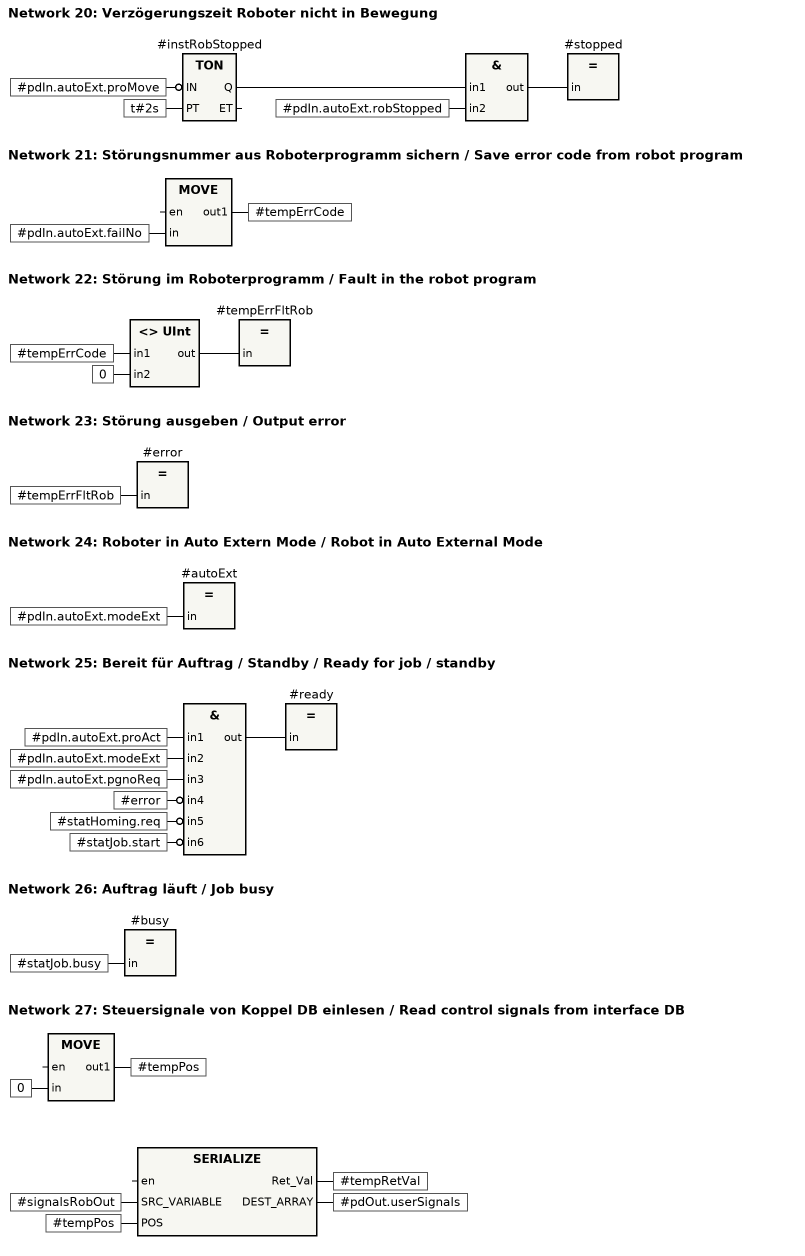
   #instRobStopped(IN := NOT #pdIn.autoExt.proMove, PT := t#2s);   // TON
   #stopped := #instRobStopped.Q AND #pdIn.autoExt.robStopped;
END_REGION

REGION Network 21: Störungsnummer aus Roboterprogramm sichern / Save error code from robot program
   #tempErrCode := #pdIn.autoExt.failNo;
END_REGION

REGION Network 22: Störung im Roboterprogramm / Fault in the robot program
   #tempErrFltRob := #tempErrCode <> 0;
END_REGION

REGION Network 23: Störung ausgeben / Output error
   #error := #tempErrFltRob;
END_REGION

REGION Network 24: Roboter in Auto Extern Mode / Robot in Auto External Mode
   #autoExt := #pdIn.autoExt.modeExt;
END_REGION

REGION Network 25: Bereit für Auftrag / Standby / Ready for job / standby
   #ready := #pdIn.autoExt.proAct AND #pdIn.autoExt.modeExt AND #pdIn.autoExt.pgnoReq AND NOT #error AND NOT #statHoming.req AND NOT #statJob.start;
END_REGION

REGION Network 26: Auftrag läuft / Job busy
   #busy := #statJob.busy;
END_REGION

REGION Network 27: Steuersignale von Koppel DB einlesen / Read control signals from interface DB
   // no SCL statement known for Serialize: written as a call
   #tempPos := 0;
   #tempRetVal := Serialize(SRC_VARIABLE := #signalsRobOut, POS := #tempPos, DEST_ARRAY => #pdOut.userSignals);
END_REGION

REGION Network 28: Peripherie schreiben / Write periphery
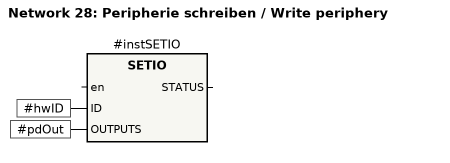
   #instSETIO(ID := #hwID, OUTPUTS := #pdOut);   // SETIO
END_REGION
END_FUNCTION_BLOCK

// folder: 9. Library/9.2 Actors/9.9.9 Simulation

FUNCTION_BLOCK "Actor2Ins2OutsSim"   // FB9991, FBD
TITLE = Aktoransteuerung 2 Ins / 2 Outs
{ S7_Optimized_Access := 'TRUE' }
VERSION : 0.1
// Ersteller: Andreas Fast Automation
// E-Mail: automation@fast-andreas.de
// 
// Projekt dient zu Demonstrationszwecken und frei genutzt werden.
// 
// Bausteinbeschreibung:
   VAR_INPUT
      iudtSimInterface : "typeSimInterface";
      ixHomePos : Bool;
      ixWorkPos : Bool;
   END_VAR
   VAR_IN_OUT
      qxHomePos : Bool;
      qxWorkPos : Bool;
      iqudtCtrl : Struct
         setHomePos : Bool;
         setWorkPos : Bool;
         isInHomePos : Bool;
         isInWorkPos : Bool;
      END_STRUCT;
      iqbSimIntAktor : Byte;   // Bit 0 = i_HomePos; Bit 1 = i_WorkPos; Bit 2 = q_SetHome; Bit 3 = q_SetWork
   END_VAR
   VAR
      sudtSimIntAktor : "typeSimAktor2Ins2Outs";
      sxSimDeactivatedFlag : Bool;
      sxSimDeactivated : Bool;
   END_VAR
   VAR_TEMP
      retVal : Int;
      tmpGrundstellungPhysikalisch : Bool;
      "tmpGrundstellungPhysikalisch+Virtuell" : Bool;
      tmpGrundstellungNurVirtuell : Bool;
   END_VAR
   VAR_TEMP   // added for the SCL form of the ladder/FBD networks
      _w1 : Bool;
      _w2 : Bool;
   END_VAR
BEGIN

REGION Network 1: Erkennung Simulation wird abgeschaltet
   // Wenn die Simulation abgeschaltet wird, sollen die physikalischen Ausgänge ihre aktuellen Zustände behalten um mögliche ungewollte Maschinenzustände zu vermeiden.
   // Das bedeutet, bei Abschaltung der Simulation werden die Ansteuerbefehle im "iqudtCtrl" and die physikalischen Ansteuerungen angepasst.
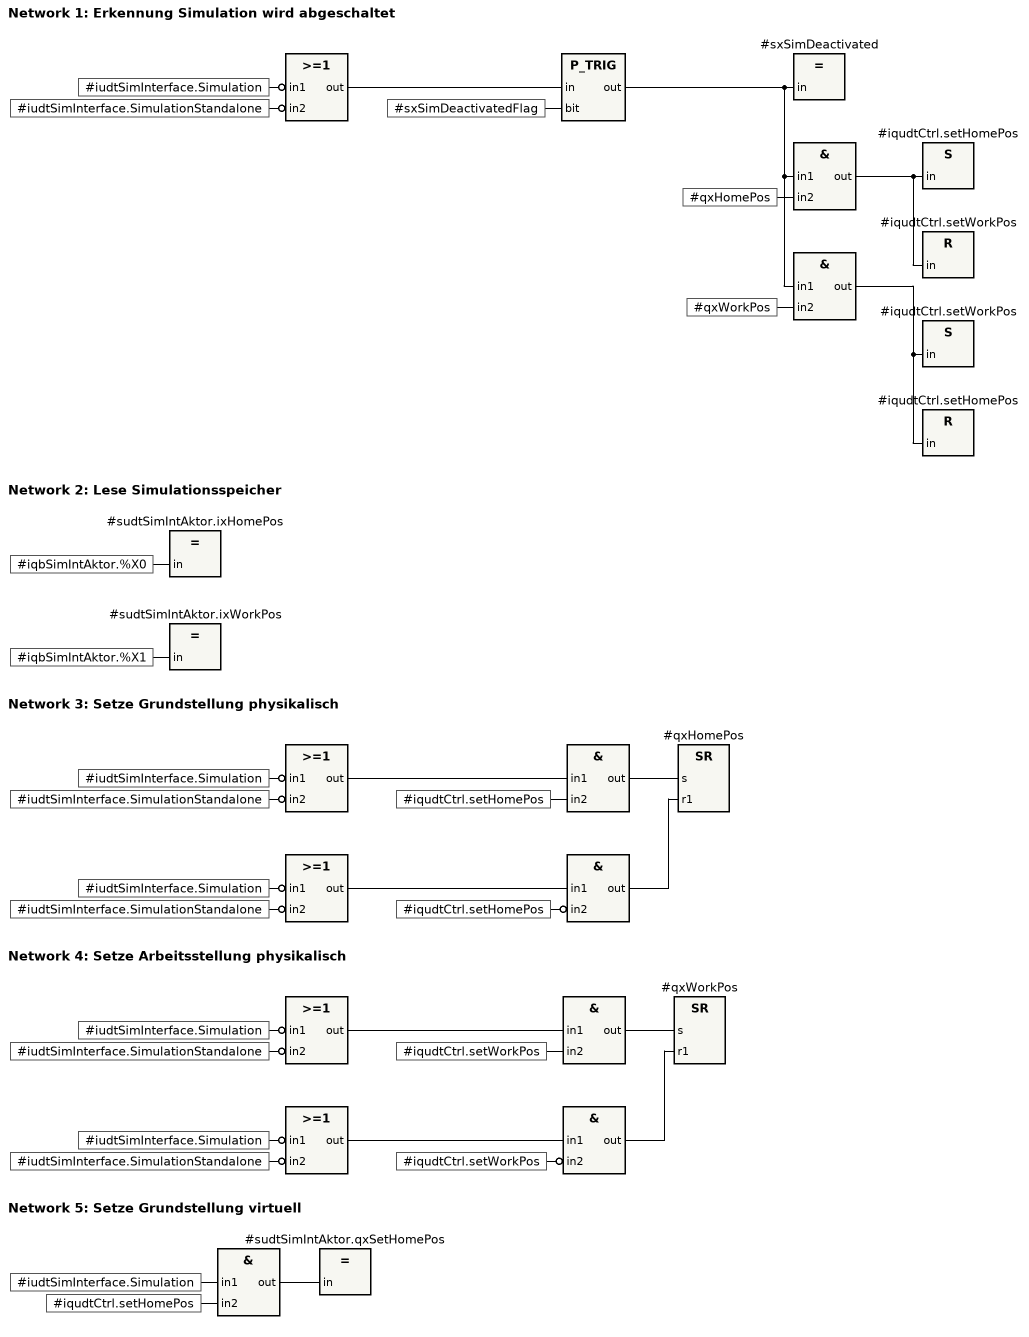
   #_w1 := NOT #iudtSimInterface.Simulation OR NOT #iudtSimInterface.SimulationStandalone;
   #_w2 := #_w1 AND NOT #sxSimDeactivatedFlag;   // rising edge
   #sxSimDeactivatedFlag := #_w1;
   #sxSimDeactivated := #_w2;
   IF #_w2 AND #qxHomePos THEN
       #iqudtCtrl.setHomePos := TRUE;
       #iqudtCtrl.setWorkPos := FALSE;
   END_IF;
   IF #_w2 AND #qxWorkPos THEN
       #iqudtCtrl.setWorkPos := TRUE;
       #iqudtCtrl.setHomePos := FALSE;
   END_IF;
END_REGION

REGION Network 2: Lese Simulationsspeicher
   #sudtSimIntAktor.ixHomePos := #iqbSimIntAktor.%X0;
   #sudtSimIntAktor.ixWorkPos := #iqbSimIntAktor.%X1;
END_REGION

REGION Network 3: Setze Grundstellung physikalisch
   IF (NOT #iudtSimInterface.Simulation OR NOT #iudtSimInterface.SimulationStandalone) AND #iqudtCtrl.setHomePos THEN
       #qxHomePos := TRUE;   // SR flip-flop
   END_IF;
   IF (NOT #iudtSimInterface.Simulation OR NOT #iudtSimInterface.SimulationStandalone) AND NOT #iqudtCtrl.setHomePos THEN
       #qxHomePos := FALSE;
   END_IF;
END_REGION

REGION Network 4: Setze Arbeitsstellung physikalisch
   IF (NOT #iudtSimInterface.Simulation OR NOT #iudtSimInterface.SimulationStandalone) AND #iqudtCtrl.setWorkPos THEN
       #qxWorkPos := TRUE;   // SR flip-flop
   END_IF;
   IF (NOT #iudtSimInterface.Simulation OR NOT #iudtSimInterface.SimulationStandalone) AND NOT #iqudtCtrl.setWorkPos THEN
       #qxWorkPos := FALSE;
   END_IF;
END_REGION

REGION Network 5: Setze Grundstellung virtuell
   #sudtSimIntAktor.qxSetHomePos := #iudtSimInterface.Simulation AND #iqudtCtrl.setHomePos;
END_REGION

REGION Network 6: Setze Arbeitsstellung virtuell
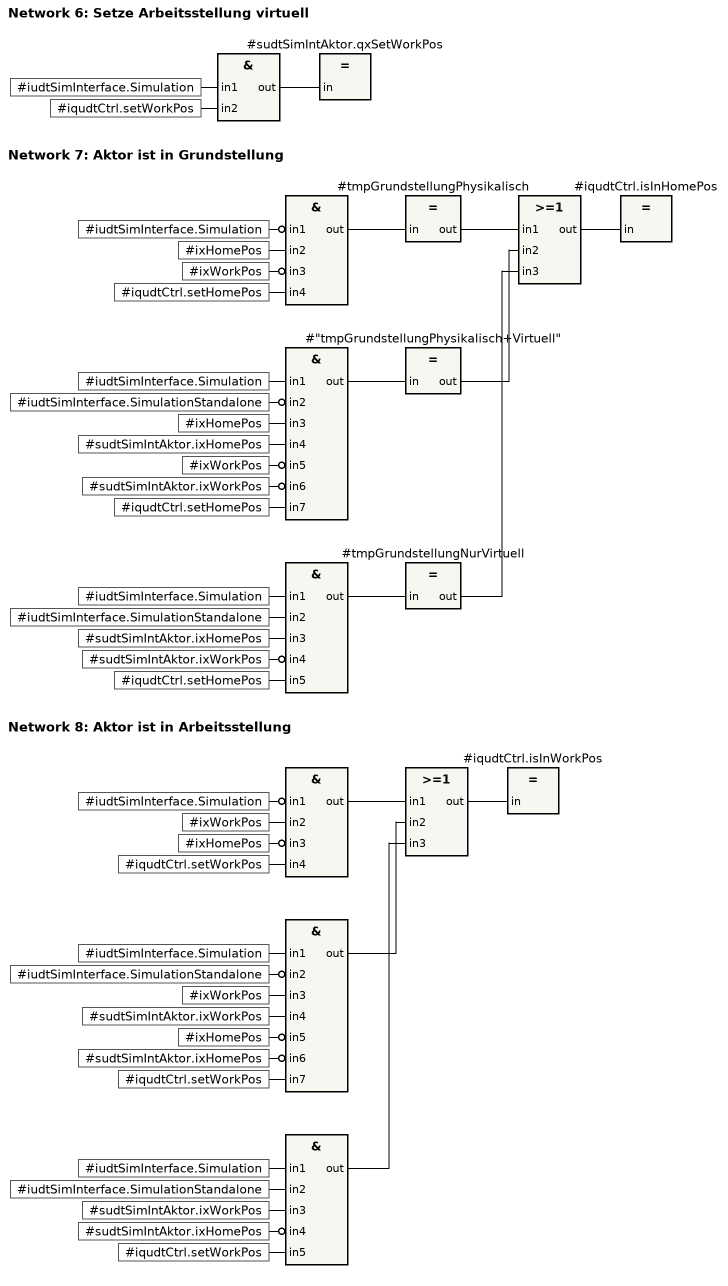
   #sudtSimIntAktor.qxSetWorkPos := #iudtSimInterface.Simulation AND #iqudtCtrl.setWorkPos;
END_REGION

REGION Network 7: Aktor ist in Grundstellung
   #tmpGrundstellungPhysikalisch := NOT #iudtSimInterface.Simulation AND #ixHomePos AND NOT #ixWorkPos AND #iqudtCtrl.setHomePos;
   #"tmpGrundstellungPhysikalisch+Virtuell" := #iudtSimInterface.Simulation AND NOT #iudtSimInterface.SimulationStandalone AND #ixHomePos AND #sudtSimIntAktor.ixHomePos AND NOT #ixWorkPos AND NOT #sudtSimIntAktor.ixWorkPos AND #iqudtCtrl.setHomePos;
   #tmpGrundstellungNurVirtuell := #iudtSimInterface.Simulation AND #iudtSimInterface.SimulationStandalone AND #sudtSimIntAktor.ixHomePos AND NOT #sudtSimIntAktor.ixWorkPos AND #iqudtCtrl.setHomePos;
   #iqudtCtrl.isInHomePos := #tmpGrundstellungPhysikalisch OR #"tmpGrundstellungPhysikalisch+Virtuell" OR #tmpGrundstellungNurVirtuell;
END_REGION

REGION Network 8: Aktor ist in Arbeitsstellung
   #iqudtCtrl.isInWorkPos := (NOT #iudtSimInterface.Simulation AND #ixWorkPos AND NOT #ixHomePos AND #iqudtCtrl.setWorkPos) OR (#iudtSimInterface.Simulation AND NOT #iudtSimInterface.SimulationStandalone AND #ixWorkPos AND #sudtSimIntAktor.ixWorkPos AND NOT #ixHomePos AND NOT #sudtSimIntAktor.ixHomePos AND #iqudtCtrl.setWorkPos) OR (#iudtSimInterface.Simulation AND #iudtSimInterface.SimulationStandalone AND #sudtSimIntAktor.ixWorkPos AND NOT #sudtSimIntAktor.ixHomePos AND #iqudtCtrl.setWorkPos);
END_REGION

REGION Network 9: Schreibe Aktorbefehle zur Simulation
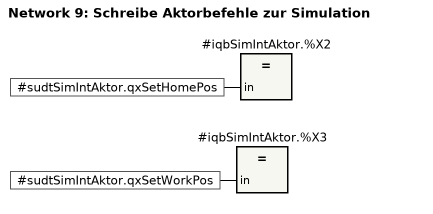
   #iqbSimIntAktor.%X2 := #sudtSimIntAktor.qxSetHomePos;
   #iqbSimIntAktor.%X3 := #sudtSimIntAktor.qxSetWorkPos;
END_REGION
END_FUNCTION_BLOCK

// folder: 9. Library/9.3 Processes

FUNCTION_BLOCK "Process_Stopper"   // FB9301, FBD
TITLE = Steuerung eines Stoppers
{ S7_Optimized_Access := 'TRUE' }
VERSION : 0.1
   VAR_INPUT
      ixBypass : Bool;   // UP umgehen / beenden
      ixStopperClosed : Bool;   // Stopper ist geschlossen/oben
      ixCarrierPresent : Bool;   // WT am Stopper vorhanden
      ixTargetReached : Bool := true;   // WT-Sensor des nächsten Ziels (falls nicht vorhanden muss dieser Eingang "true" sein)
      ixStop : Bool;   // Stoppt Ablauf / Schließt wieder den Stopper (z.B. bei einer Störung ausserhalb)
      itStopperRelease : Time := T#50ms;   // Zusätzliche Verzögerungszeit für Stopper öffnen, nachdem WT den Stopper verlassen hat
      itMaxRuntime : Time := t#5s;   // Maximale Laufzeit für diesen Prozess
   END_VAR
   VAR_OUTPUT
      qxSeqActive : Bool;   // Stopperablauf ist aktiv
      qxIsInHome : Bool;   // Ist in Grundstellung
      qxStopperOpen : Bool;   // Stopper öffnen
      qxError : Bool;   // Sammelstörung
      qbErrorCode : Byte;   // Ausgabe Fehlercode (siehe Sammelstörung Netzwerkkommentar)
   END_VAR
   VAR_IN_OUT
      signals : "typeStationSignals";   // Stationssignale
      iqxRequest : Bool;   // 1 = Starte Ablauf (wird nach Ausführung intern zurückgesetzt)
   END_VAR
   VAR
      sinstTonStopperOpened : TON_TIME;
      sinstTonStopperBusyError : TON_TIME;
      sinstTonMaxRuntime : TON_TIME;
      sxStep1 : Bool;
      sxStep2 : Bool;
      sxStep3 : Bool;
      sxCheckWtIsGone : Bool;   // Prüfe, ob WT den Stopper verlassen hat
   END_VAR
   VAR_TEMP
      txWT_Error_1 : Bool;
      txWT_Error_2 : Bool;
      txWT_Error_3 : Bool;
      txWT_Error_4 : Bool;
      txWT_Error_5 : Bool;
   END_VAR
   VAR_TEMP   // added for the SCL form of the ladder/FBD networks
      _w1 : Bool;
      _w2 : Bool;
   END_VAR
BEGIN

REGION Network 1: Schritt 1: Start
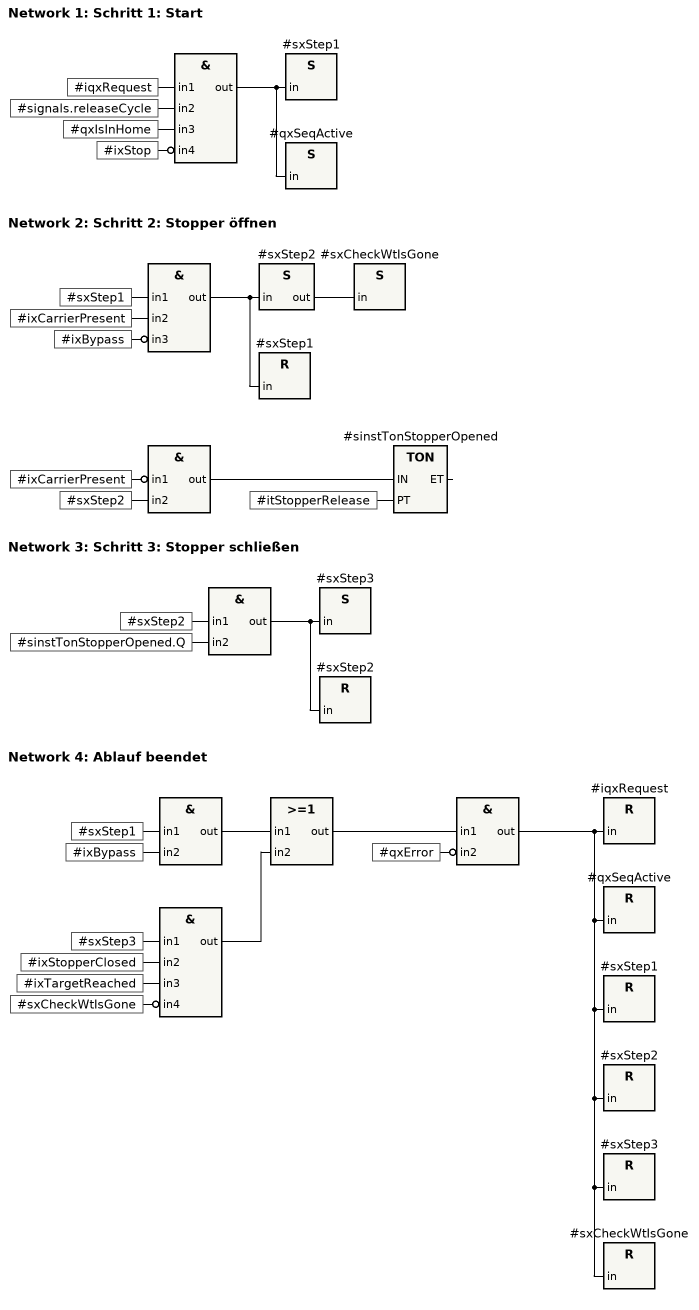
   IF #iqxRequest AND #signals.releaseCycle AND #qxIsInHome AND NOT #ixStop THEN
       #sxStep1 := TRUE;
       #qxSeqActive := TRUE;
   END_IF;
END_REGION

REGION Network 2: Schritt 2: Stopper öffnen
   IF #sxStep1 AND #ixCarrierPresent AND NOT #ixBypass THEN
       #sxStep2 := TRUE;
       #sxCheckWtIsGone := TRUE;
       #sxStep1 := FALSE;
   END_IF;
   #sinstTonStopperOpened(IN := NOT #ixCarrierPresent AND #sxStep2, PT := #itStopperRelease);   // TON
END_REGION

REGION Network 3: Schritt 3: Stopper schließen
   IF #sxStep2 AND #sinstTonStopperOpened.Q THEN
       #sxStep3 := TRUE;
       #sxStep2 := FALSE;
   END_IF;
END_REGION

REGION Network 4: Ablauf beendet
   IF ((#sxStep1 AND #ixBypass) OR (#sxStep3 AND #ixStopperClosed AND #ixTargetReached AND NOT #sxCheckWtIsGone)) AND NOT #qxError THEN
       #iqxRequest := FALSE;
       #qxSeqActive := FALSE;
   END_IF;
   #_w1 := ((#sxStep1 AND #ixBypass) OR (#sxStep3 AND #ixStopperClosed AND #ixTargetReached AND NOT #sxCheckWtIsGone)) AND NOT #qxError;
   IF #_w1 THEN
       #sxStep1 := FALSE;
       #sxStep2 := FALSE;
       #sxStep3 := FALSE;
       #sxCheckWtIsGone := FALSE;
   END_IF;
END_REGION

REGION Network 5: Reset
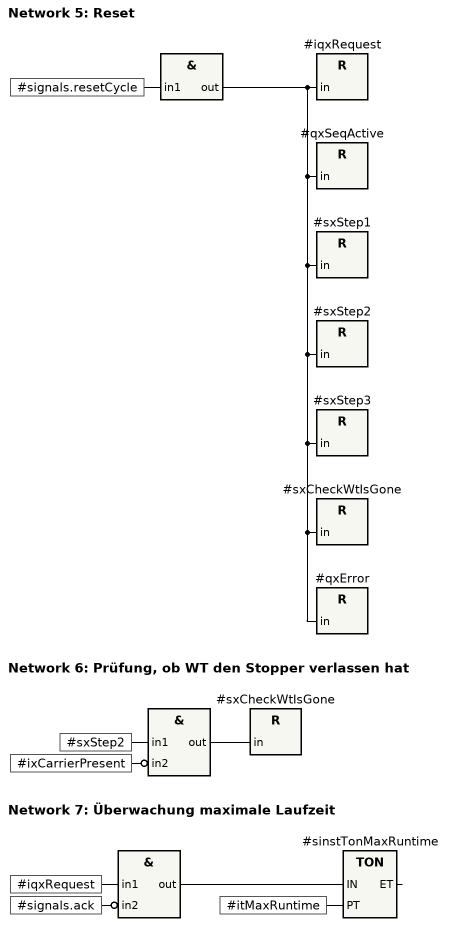
   IF #signals.resetCycle THEN
       #iqxRequest := FALSE;
       #qxSeqActive := FALSE;
       #sxStep1 := FALSE;
       #sxStep2 := FALSE;
       #sxStep3 := FALSE;
       #sxCheckWtIsGone := FALSE;
       #qxError := FALSE;
   END_IF;
END_REGION

REGION Network 6: Prüfung, ob WT den Stopper verlassen hat
   IF #sxStep2 AND NOT #ixCarrierPresent THEN #sxCheckWtIsGone := FALSE; END_IF;
END_REGION

REGION Network 7: Überwachung maximale Laufzeit
   #sinstTonMaxRuntime(IN := #iqxRequest AND NOT #signals.ack, PT := #itMaxRuntime);   // TON
END_REGION

REGION Network 8: Sammelstörung
   // 1. Kein WT am Stopper vorhanden
   // 2. Fehler, WT hat den Stopper nicht verlassen 
   // 3. WT hat den nächsten Stopper innerhalb der maximalen Laufzeit nicht erreicht
   // 4. Maximale Laufzeit überschritten
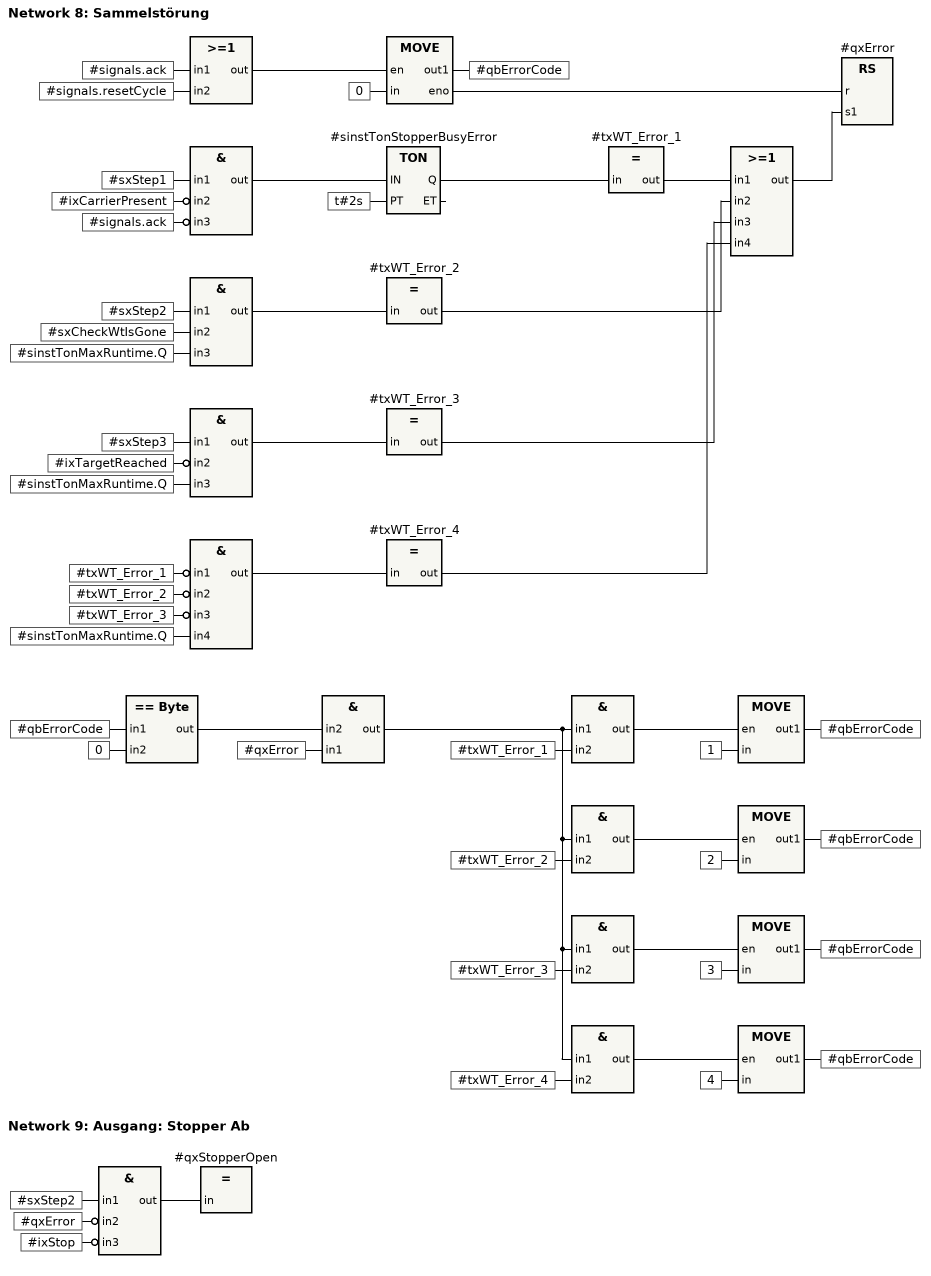
   #_w1 := #signals.ack OR #signals.resetCycle;
   IF #_w1 THEN #qbErrorCode := 0; END_IF;
   #sinstTonStopperBusyError(IN := #sxStep1 AND NOT #ixCarrierPresent AND NOT #signals.ack, PT := t#2s);   // TON
   #txWT_Error_1 := #sinstTonStopperBusyError.Q;
   #txWT_Error_2 := #sxStep2 AND #sxCheckWtIsGone AND #sinstTonMaxRuntime.Q;
   #txWT_Error_3 := #sxStep3 AND NOT #ixTargetReached AND #sinstTonMaxRuntime.Q;
   #txWT_Error_4 := NOT #txWT_Error_1 AND NOT #txWT_Error_2 AND NOT #txWT_Error_3 AND #sinstTonMaxRuntime.Q;
   IF #_w1 THEN
       #qxError := FALSE;   // RS flip-flop
   END_IF;
   IF #sinstTonStopperBusyError.Q OR #txWT_Error_2 OR #txWT_Error_3 OR #txWT_Error_4 THEN
       #qxError := TRUE;
   END_IF;
   #_w2 := (#qbErrorCode = 0) AND #qxError;
   IF #_w2 AND #txWT_Error_1 THEN #qbErrorCode := 1; END_IF;
   IF #_w2 AND #txWT_Error_2 THEN #qbErrorCode := 2; END_IF;
   IF #_w2 AND #txWT_Error_3 THEN #qbErrorCode := 3; END_IF;
   IF #_w2 AND #txWT_Error_4 THEN #qbErrorCode := 4; END_IF;
END_REGION

REGION Network 9: Ausgang: Stopper Ab
   #qxStopperOpen := #sxStep2 AND NOT #qxError AND NOT #ixStop;
END_REGION

REGION Network 10: Steht in Grundstellung
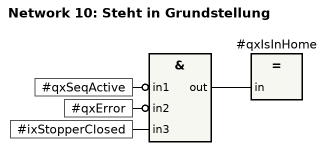
   #qxIsInHome := NOT #qxSeqActive AND NOT #qxError AND #ixStopperClosed;
END_REGION
END_FUNCTION_BLOCK

FUNCTION_BLOCK "Sq_Process_Stopper"   // FB9302, GRAPH_PLUS
{ S7_Optimized_Access := 'TRUE' }
VERSION : 0.1
   VAR_INPUT
      OFF_SQ : Bool := false;   // Kette ausschalten
      INIT_SQ : Bool := false;   // Kette in Initialzustand versetzen
      ACK_EF : Bool := false;   // Alle Fehler und Störungen quittieren
      S_PREV : Bool := false;   // Vorherigen Schritt am Parameter S_NO ausgeben
      S_NEXT : Bool := false;   // Nächsten Schritt am Parameter S_NO anzeigen
      SW_AUTO : Bool := false;   // Automatischer Betrieb
      SW_TAP : Bool := false;   // Halbautomatisch/Weiterschalten mit Transition
      SW_TOP : Bool := false;   // Halbautomatisch/Ignoriere Transition
      SW_MAN : Bool := false;   // Handbetrieb
      S_SEL : Int := 0;   // Schritt auswählen, der an S_NO ausgegeben werden soll
      S_ON : Bool := false;   // Schritt aktivieren, der an Parameter S_NO anliegt
      S_OFF : Bool := false;   // Schritt deaktivieren, der an Parameter S_NO anliegt
      T_PUSH : Bool := false;   // Schaltfreigabe für Transition im halbautomatischen Betrieb
      ixStart : Bool;   // Startfreigabe
      ixCarrierPresent : Bool;   // WT am Stopper vorhanden
      ixCheckTargetReached : Bool := false;   // 0 = Keine Sensor-Zielüberwachung nach Lift vorhanden
      ixTargetReached : Bool := false;   // WT-Sensor des nächsten Ziels
      itStopperRelease : Time := T#50ms;   // Zusätzliche Verzögerungszeit für Stopper öffnen, nachdem WT den Stopper verlassen hat
      itMaxRuntime : Time := t#5s;   // Maximale Laufzeit für diesen Prozess
   END_VAR
   VAR_OUTPUT
      S_NO : Int := 0;   // Schrittnummer
      S_MORE : Bool := false;   // Weitere Schritte sind vorhanden und können in S_NO angezeigt werden.
      S_ACTIVE : Bool := false;   // Schritt, der an Parameter S_NO angezeigt wird, ist aktiv
      ERR_FLT : Bool := false;   // Sammelfehler Interlock oder Supervision
      AUTO_ON : Bool := false;   // Automatischer Betrieb eingeschaltet
      TAP_ON : Bool := false;   // Halbautomatischer Betrieb/Schritt mit Transition eingeschaltet
      TOP_ON : Bool := false;   // Halbautomatischer Betrieb/Ignoriere Transition eingeschaltet
      MAN_ON : Bool := false;   // Handbetrieb eingeschaltet
      qxWaitForTarget : Bool;   // Warte bis Ziel erreicht
      qxIsActive : Bool;   // Process läuft
      qxIsInHome : Bool;   // steht in Grundstellung
   END_VAR
   VAR_IN_OUT
      signals : "typeStationSignals";   // Stationssteuersignale
      sq : "typeStepSequence";   // Schrittkettensteuersignale
      cylinder_stopper : "typeActor_1Out1In";   // Aktor für den Stopper
   END_VAR
   VAR
      sstReleaseCycle : Struct
         ErrorAck : Bool;
         No_LastCycle : Int;
         T : Time;   // Aktive Zeit des ReleaseCycle
         Tck : Time;
         TckPrev : Time;
      END_STRUCT;
      HMI_INFO : Array[0..8] of UInt;
      IF_PAR : G7_IfParPlus_V6;
      RT_DATA : G7_RTDataPlus_V6;   // Interner Datenbereich
      Automatikablauf : G7_TransitionPlus_V6;   // Transitionsstruktur
      Freigabe : G7_TransitionPlus_V6;   // Transitionsstruktur
      Trans3 : G7_TransitionPlus_V6;   // Transitionsstruktur
      Fertig : G7_TransitionPlus_V6;   // Transitionsstruktur
      Grundstellungsfahrt : G7_TransitionPlus_V6;   // Transitionsstruktur
      GST_Aktiv : G7_TransitionPlus_V6;   // Transitionsstruktur
      GST_Beendet : G7_TransitionPlus_V6;   // Transitionsstruktur
      Beendet : G7_TransitionPlus_V6;   // Transitionsstruktur
      "WT hat Stopper verlassen" : G7_TransitionPlus_V6;   // Transitionsstruktur / Transition structure
      "Nachlaufzeit abgelaufen" : G7_TransitionPlus_V6;   // Transitionsstruktur / Transition structure
      "Ziel erreicht" : G7_TransitionPlus_V6;   // Transitionsstruktur / Transition structure
      Initialschritt : G7_StepPlus_V6;   // Schrittstruktur
      Grundstellung : G7_StepPlus_V6;   // Schrittstruktur
      SK_läuft : G7_StepPlus_V6;   // Schrittstruktur
      Fertigmeldung : G7_StepPlus_V6;   // Schrittstruktur
      "Start Grundstellungsfahrt" : G7_StepPlus_V6;   // Schrittstruktur
      "Fertig Grundstellungsfahrt" : G7_StepPlus_V6;   // Schrittstruktur
      Ende : G7_StepPlus_V6;   // Schrittstruktur
      "Stopper öffnen" : G7_StepPlus_V6;   // Schrittstruktur / Step structure
      Nachlaufzeit : G7_StepPlus_V6;   // Schrittstruktur / Step structure
      WaitForTarget : G7_StepPlus_V6;   // Schrittstruktur / Step structure
      SINI : Array[0..1] of USInt;
      LSTT : Array[0..10] of USInt;
      ATAJ : Array[0..10] of USInt;
      ATAB : Array[0..10] of USInt;
      PSTT : Array[0..10] of USInt;
      NSTT : Array[0..10] of USInt;
      ASSJ : Array[0..9] of USInt;
      ASSB : Array[0..9] of USInt;
      PTTS : Array[0..9] of USInt;
      NTTS : Array[0..9] of USInt;
      SW_SQTS : Array[0..9] of USInt;
      SWITCH : Array[0..1] of USInt;
      TVX : Array[0..3] of USInt;
      TTX : Array[0..3] of USInt;
      TSX : Array[0..1] of USInt;
      S00X : Array[0..1] of USInt;
      SOFFX : Array[0..1] of USInt;
      SONX : Array[0..1] of USInt;
      SAX : Array[0..1] of USInt;
      SERRX : Array[0..10] of USInt;
      SMX : Array[0..10] of USInt;
      S0X : Array[0..10] of USInt;
      S1X : Array[0..10] of USInt;
      IL_ALARM_INST : Diag_Alarm;
      SUP_ALARM_INST : Diag_Alarm;
      STEP_TIME_ALARM_INST : Diag_Alarm;
      IEC_TIMER_INST : IEC_TIMER;
      TRANSACTION_FLAG : Bool := false;
   END_VAR
   VAR_TEMP
      txStartCondition : Bool;
      tdTckDiff : DInt;
   END_VAR
   VAR_TEMP   // added for the SCL form of the ladder/FBD networks
      _w1 : Bool;
   END_VAR
   // SINI[0] := 2;
   // LSTT[0] := 255;
   // LSTT[1] := 255;
   // LSTT[2] := 255;
   // LSTT[3] := 255;
   // LSTT[4] := 255;
   // LSTT[5] := 255;
   // LSTT[6] := 255;
   // LSTT[7] := 1;
   // ATAJ[1] := 1;
   // ATAJ[2] := 2;
   // ATAJ[3] := 6;
   // ATAJ[4] := 4;
   // ATAJ[5] := 5;
   // ATAJ[6] := 3;
   // ATAJ[7] := 7;
   // ATAB[0] := 4;
   // ATAB[1] := 1;
   // ATAB[2] := 2;
   // ATAB[3] := 3;
   // ATAB[5] := 5;
   // ATAB[6] := 6;
   // ATAB[7] := 7;
   // PSTT[1] := 1;
   // PSTT[2] := 2;
   // PSTT[3] := 3;
   // PSTT[5] := 4;
   // PSTT[6] := 5;
   // PSTT[7] := 6;
   // NSTT[0] := 1;
   // NSTT[1] := 2;
   // NSTT[2] := 7;
   // NSTT[3] := 6;
   // NSTT[4] := 4;
   // NSTT[5] := 5;
   // NSTT[6] := 6;
   // NSTT[7] := 1;
   // ASSJ[1] := 1;
   // ASSJ[2] := 2;
   // ASSJ[3] := 3;
   // ASSJ[4] := 4;
   // ASSJ[5] := 5;
   // ASSJ[6] := 6;
   // ASSB[1] := 1;
   // ASSB[2] := 2;
   // ASSB[3] := 3;
   // ASSB[4] := 4;
   // ASSB[5] := 5;
   // ASSB[6] := 6;
   // PTTS[0] := 255;
   // PTTS[2] := 1;
   // PTTS[3] := 10;
   // PTTS[4] := 4;
   // PTTS[5] := 5;
   // PTTS[6] := 3;
   // NTTS[1] := 1;
   // NTTS[2] := 2;
   // NTTS[3] := 3;
   // NTTS[4] := 5;
   // NTTS[5] := 6;
   // NTTS[6] := 7;
   // SW_SQTS[1] := 1;
   // SW_SQTS[2] := 1;
   // SW_SQTS[3] := 1;
   // SW_SQTS[4] := 2;
   // SW_SQTS[5] := 2;
   // SW_SQTS[6] := 3;
   // TVX[0] := 16#1;
   // TTX[0] := 16#1;
   // TSX[0] := 16#1;
   // S00X[0] := 16#1;
   // SOFFX[0] := 16#1;
   // SONX[0] := 16#1;
   // SAX[0] := 16#1;
   // SERRX[0] := 16#1;
   // SMX[0] := 16#1;
   // S0X[0] := 16#1;
   // S1X[0] := 16#1;
   // LSTT[8] := 255;
   // ATAJ[8] := 8;
   // ATAB[8] := 8;
   // PSTT[8] := 7;
   // NSTT[8] := 8;
   // ASSJ[7] := 7;
   // ASSB[7] := 7;
   // PTTS[7] := 2;
   // NTTS[7] := 8;
   // SW_SQTS[7] := 1;
   // LSTT[9] := 255;
   // LSTT[10] := 255;
   // ATAJ[9] := 9;
   // ATAJ[10] := 10;
   // ATAB[9] := 9;
   // ATAB[10] := 10;
   // PSTT[9] := 8;
   // PSTT[10] := 9;
   // NSTT[9] := 9;
   // NSTT[10] := 3;
   // ASSJ[8] := 8;
   // ASSJ[9] := 9;
   // ASSB[8] := 8;
   // ASSB[9] := 9;
   // PTTS[8] := 8;
   // PTTS[9] := 9;
   // NTTS[8] := 9;
   // NTTS[9] := 10;
   // SW_SQTS[8] := 1;
   // SW_SQTS[9] := 1;
BEGIN
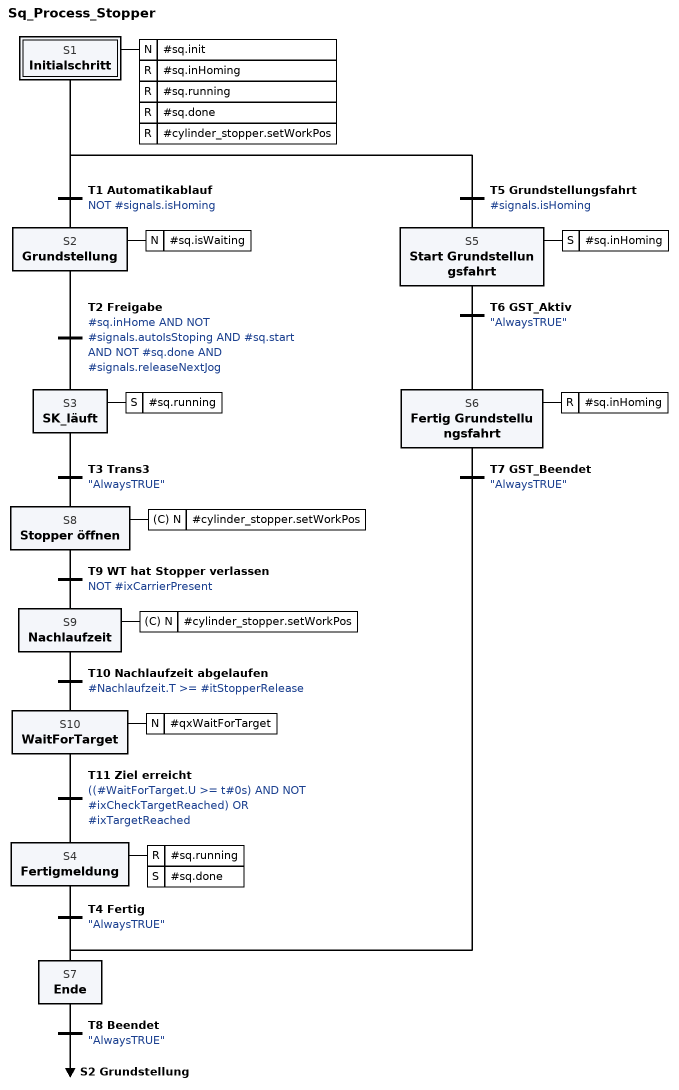
   // permanent pre-instructions
   NETWORK 1
   TITLE = Schrittkette verfügbar
      #sq.exists := true;
   NETWORK 2
   TITLE = Schrittkette in Grundstellung (Erweitern)
      #sq.inHome := #Grundstellung.X AND #cylinder_stopper.inHomePos;
   NETWORK 3
   TITLE = Startbedingung (Erweitern)
      #txStartCondition := (NOT #ixCheckTargetReached OR NOT #ixTargetReached) AND #ixStart AND #ixCarrierPresent;
   NETWORK 4
   TITLE = Schrittkette starten
      #sq.start := #sq.inHome AND NOT #sq.running AND #signals.releaseCycle AND NOT #signals.isHoming AND #txStartCondition;
      IF #sq.start THEN #sq.done := FALSE; END_IF;
   NETWORK 5
   TITLE = ReleaseCycle Timer
      // ENO of a box is taken as its EN; it also drops when the box reports an error
      #_w1 := #ACK_EF AND NOT #sstReleaseCycle.ErrorAck;   // rising edge
      #sstReleaseCycle.ErrorAck := #ACK_EF;
      IF (#S_NO <> #sstReleaseCycle.No_LastCycle) OR #_w1 THEN
          #sstReleaseCycle.T := T#0MS;
          #sstReleaseCycle.TckPrev := #sstReleaseCycle.Tck;
          #sstReleaseCycle.No_LastCycle := #S_NO;
      END_IF;
      #sstReleaseCycle.Tck := TIME_TCK();
      #tdTckDiff := #sstReleaseCycle.Tck - #sstReleaseCycle.TckPrev;
      #sstReleaseCycle.TckPrev := #sstReleaseCycle.Tck;
      IF (0 <= #tdTckDiff) AND (#tdTckDiff <= 1000) AND #signals.releaseCycle THEN
          #sstReleaseCycle.T := #sstReleaseCycle.T + #tdTckDiff;
      END_IF;

   // sequencer 1
   INITIAL_STEP Initialschritt:   // S1, max time T#10S, warning time T#7S
              N    #sq.init
              R    #sq.inHoming
              R    #sq.running
              R    #sq.done
              R    #cylinder_stopper.setWorkPos
   END_STEP
   TRANSITION Automatikablauf FROM Initialschritt TO Grundstellung   // T1
      := NOT #signals.isHoming;
   END_TRANSITION
   TRANSITION Grundstellungsfahrt FROM Initialschritt TO "Start Grundstellungsfahrt"   // T5
      := #signals.isHoming;
   END_TRANSITION
   STEP Grundstellung:   // S2, max time T#10S, warning time T#7S
              N    #sq.isWaiting
   END_STEP
   TRANSITION Freigabe FROM Grundstellung TO SK_läuft   // T2
      := #sq.inHome AND NOT #signals.autoIsStoping AND #sq.start AND NOT #sq.done AND #signals.releaseNextJog;
   END_TRANSITION
   STEP SK_läuft:   // S3, max time T#10S, warning time T#7S
              S    #sq.running
   END_STEP
   TRANSITION Trans3 FROM SK_läuft TO "Stopper öffnen"   // T3
      := "AlwaysTRUE";
   END_TRANSITION
   STEP Fertigmeldung:   // S4, max time T#10S, warning time T#7S
              R    #sq.running
              S    #sq.done
   END_STEP
   TRANSITION Fertig FROM Fertigmeldung TO Ende   // T4
      := "AlwaysTRUE";
   END_TRANSITION
   STEP "Start Grundstellungsfahrt":   // S5, max time T#10S, warning time T#7S
              S    #sq.inHoming
   END_STEP
   TRANSITION GST_Aktiv FROM "Start Grundstellungsfahrt" TO "Fertig Grundstellungsfahrt"   // T6
      := "AlwaysTRUE";
   END_TRANSITION
   STEP "Fertig Grundstellungsfahrt":   // S6, max time T#10S, warning time T#7S
              R    #sq.inHoming
   END_STEP
   TRANSITION GST_Beendet FROM "Fertig Grundstellungsfahrt" TO Ende   // T7
      := "AlwaysTRUE";
   END_TRANSITION
   STEP Ende:   // S7, max time T#10S, warning time T#7S
   END_STEP
   TRANSITION Beendet FROM Ende TO Grundstellung   // T8, jump
      := "AlwaysTRUE";
   END_TRANSITION
   STEP "Stopper öffnen":   // S8, max time T#10S, warning time T#7S
      supervision V := ((#sstReleaseCycle.T >= #itMaxRuntime) AND false) OR (#cylinder_stopper.inError AND #"Stopper öffnen".X AND false);
      (C)     N    #cylinder_stopper.setWorkPos
   END_STEP
   TRANSITION "WT hat Stopper verlassen" FROM "Stopper öffnen" TO Nachlaufzeit   // T9
      := NOT #ixCarrierPresent;
   END_TRANSITION
   STEP Nachlaufzeit:   // S9, max time T#10S, warning time T#7S
      (C)     N    #cylinder_stopper.setWorkPos
   END_STEP
   TRANSITION "Nachlaufzeit abgelaufen" FROM Nachlaufzeit TO WaitForTarget   // T10
      := #Nachlaufzeit.T >= #itStopperRelease;
   END_TRANSITION
   STEP WaitForTarget:   // S10, max time T#10S, warning time T#7S
      supervision V := #sstReleaseCycle.T >= #itMaxRuntime;
              N    #qxWaitForTarget
   END_STEP
   TRANSITION "Ziel erreicht" FROM WaitForTarget TO Fertigmeldung   // T11
      := ((#WaitForTarget.U >= t#0s) AND NOT #ixCheckTargetReached) OR #ixTargetReached;
   END_TRANSITION

   // permanent post-instructions
   NETWORK 1
   TITLE = Störungssignal weitergeben
      #sq.error := #ERR_FLT;
   NETWORK 2
   TITLE = Ablauf ist aktiv
      #qxIsActive := #sq.running;
   NETWORK 3
   TITLE = steht in Grundstellung
      #qxIsInHome := #sq.inHome AND NOT #sq.running;
END_FUNCTION_BLOCK

FUNCTION_BLOCK "Sq_Process_Lift"   // FB9303, GRAPH_PLUS
{ S7_Optimized_Access := 'TRUE' }
VERSION : 0.1
   VAR_INPUT
      OFF_SQ : Bool := false;   // Kette ausschalten
      INIT_SQ : Bool := false;   // Kette in Initialzustand versetzen
      ACK_EF : Bool := false;   // Alle Fehler und Störungen quittieren
      S_PREV : Bool := false;   // Vorherigen Schritt am Parameter S_NO ausgeben
      S_NEXT : Bool := false;   // Nächsten Schritt am Parameter S_NO anzeigen
      SW_AUTO : Bool := false;   // Automatischer Betrieb
      SW_TAP : Bool := false;   // Halbautomatisch/Weiterschalten mit Transition
      SW_TOP : Bool := false;   // Halbautomatisch/Ignoriere Transition
      SW_MAN : Bool := false;   // Handbetrieb
      S_SEL : Int := 0;   // Schritt auswählen, der an S_NO ausgegeben werden soll
      S_ON : Bool := false;   // Schritt aktivieren, der an Parameter S_NO anliegt
      S_OFF : Bool := false;   // Schritt deaktivieren, der an Parameter S_NO anliegt
      T_PUSH : Bool := false;   // Schaltfreigabe für Transition im halbautomatischen Betrieb
      ixStart : Bool := true;   // Startfreigabe
      ixCarrierPresent : Bool;   // WT auf dem Lift vorhanden
      ixCheckTargetReached : Bool := false;   // 0 = Keine Sensor-Zielüberwachung nach Lift vorhanden
      ixTargetReached : Bool := false;   // WT-Sensor des nächsten Ziels
      ixExternReqConvIn : Bool;   // Externe Anforderung Förderband Einlauf starten
      itCarrierReactionDelay : Time := T#350ms;   // Verzögerungszeit für die WT-Erkennung
      itMaxRuntime : Time := t#10s;   // Maximale Laufzeit für diesen Prozess
   END_VAR
   VAR_OUTPUT
      S_NO : Int := 0;   // Schrittnummer
      S_MORE : Bool := false;   // Weitere Schritte sind vorhanden und können in S_NO angezeigt werden.
      S_ACTIVE : Bool := false;   // Schritt, der an Parameter S_NO angezeigt wird, ist aktiv
      ERR_FLT : Bool := false;   // Sammelfehler Interlock oder Supervision
      AUTO_ON : Bool := false;   // Automatischer Betrieb eingeschaltet
      TAP_ON : Bool := false;   // Halbautomatischer Betrieb/Schritt mit Transition eingeschaltet
      TOP_ON : Bool := false;   // Halbautomatischer Betrieb/Ignoriere Transition eingeschaltet
      MAN_ON : Bool := false;   // Handbetrieb eingeschaltet
      qxIsActive : Bool;   // Schrittkette läuft
      qxIsInHome : Bool;   // steht in Grundstellung
   END_VAR
   VAR_IN_OUT
      signals : "typeStationSignals";   // Stationssteuersignale
      sq : "typeStepSequence";   // Schrittkettensteuersignale
      cylinder : "typeActor_2Out2In";   // Aktor des Zylinders für den Lift
      conveyor : "typeActor_2Out0In";   // Aktor des Förderbands für den Lift
   END_VAR
   VAR
      sstReleaseCycle : Struct
         ErrorAck : Bool;
         No_LastCycle : Int;
         T : Time;   // Aktive Zeit des ReleaseCycle
         Tck : Time;
         TckPrev : Time;
      END_STRUCT;
      sinstCarrierOnLift : TON_TIME;
      sinstCarrierLeftLift : TON_TIME;
      HMI_INFO : Array[0..8] of UInt;
      IF_PAR : G7_IfParPlus_V6;
      RT_DATA : G7_RTDataPlus_V6;   // Interner Datenbereich
      Automatikablauf : G7_TransitionPlus_V6;   // Transitionsstruktur
      Freigabe : G7_TransitionPlus_V6;   // Transitionsstruktur
      Trans3 : G7_TransitionPlus_V6;   // Transitionsstruktur
      Fertig : G7_TransitionPlus_V6;   // Transitionsstruktur
      Grundstellungsfahrt : G7_TransitionPlus_V6;   // Transitionsstruktur
      GST_Aktiv : G7_TransitionPlus_V6;   // Transitionsstruktur
      GST_Beendet : G7_TransitionPlus_V6;   // Transitionsstruktur
      Beendet : G7_TransitionPlus_V6;   // Transitionsstruktur
      "WT ist komplett auf dem Lift eingefahren" : G7_TransitionPlus_V6;   // Transitionsstruktur / Transition structure
      "WT ist komplett auf dem Lift eingefahren_1" : G7_TransitionPlus_V6;   // Transitionsstruktur / Transition structure
      "Wt hat den Lift verlassen" : G7_TransitionPlus_V6;   // Transitionsstruktur / Transition structure
      "Lift steht in Arbeitsstellung" : G7_TransitionPlus_V6;   // Transitionsstruktur / Transition structure
      "Wt hat Endziel erreicht" : G7_TransitionPlus_V6;   // Transitionsstruktur / Transition structure
      "Lift steht in Grundstellung" : G7_TransitionPlus_V6;   // Transitionsstruktur / Transition structure
      "Lift steht in Grundstellung_1" : G7_TransitionPlus_V6;   // Transitionsstruktur / Transition structure
      "Endziel ist frei" : G7_TransitionPlus_V6;   // Transitionsstruktur / Transition structure
      "Endziel ist belegt" : G7_TransitionPlus_V6;   // Transitionsstruktur / Transition structure
      JogT1 : G7_TransitionPlus_V6;   // Transitionsstruktur / Transition structure
      JogT2 : G7_TransitionPlus_V6;   // Transitionsstruktur / Transition structure
      JogT3 : G7_TransitionPlus_V6;   // Transitionsstruktur / Transition structure
      Initialschritt : G7_StepPlus_V6;   // Schrittstruktur
      Grundstellung : G7_StepPlus_V6;   // Schrittstruktur
      SK_läuft : G7_StepPlus_V6;   // Schrittstruktur
      Fertigmeldung : G7_StepPlus_V6;   // Schrittstruktur
      "Start Grundstellungsfahrt" : G7_StepPlus_V6;   // Schrittstruktur
      "Fertig Grundstellungsfahrt" : G7_StepPlus_V6;   // Schrittstruktur
      Ende : G7_StepPlus_V6;   // Schrittstruktur
      ConvIn : G7_StepPlus_V6;   // Schrittstruktur / Step structure
      GS_ConvIn : G7_StepPlus_V6;   // Schrittstruktur / Step structure
      ConvOut : G7_StepPlus_V6;   // Schrittstruktur / Step structure
      LiftToWork : G7_StepPlus_V6;   // Schrittstruktur / Step structure
      WaitConvOut : G7_StepPlus_V6;   // Schrittstruktur / Step structure
      LiftToHome : G7_StepPlus_V6;   // Schrittstruktur / Step structure
      GS_CylHome : G7_StepPlus_V6;   // Schrittstruktur / Step structure
      Warte_Endziel_frei : G7_StepPlus_V6;   // Schrittstruktur / Step structure
      JogS1 : G7_StepPlus_V6;   // Schrittstruktur / Step structure
      JogS2 : G7_StepPlus_V6;   // Schrittstruktur / Step structure
      JogS3 : G7_StepPlus_V6;   // Schrittstruktur / Step structure
      SINI : Array[0..1] of USInt;
      LSTT : Array[0..19] of USInt;
      ATAJ : Array[0..19] of USInt;
      ATAB : Array[0..19] of USInt;
      PSTT : Array[0..19] of USInt;
      NSTT : Array[0..19] of USInt;
      ASSJ : Array[0..17] of USInt;
      ASSB : Array[0..17] of USInt;
      PTTS : Array[0..17] of USInt;
      NTTS : Array[0..17] of USInt;
      SW_SQTS : Array[0..17] of USInt;
      SWITCH : Array[0..3] of USInt;
      TVX : Array[0..5] of USInt;
      TTX : Array[0..5] of USInt;
      TSX : Array[0..1] of USInt;
      S00X : Array[0..1] of USInt;
      SOFFX : Array[0..1] of USInt;
      SONX : Array[0..1] of USInt;
      SAX : Array[0..1] of USInt;
      SERRX : Array[0..18] of USInt;
      SMX : Array[0..18] of USInt;
      S0X : Array[0..18] of USInt;
      S1X : Array[0..18] of USInt;
      IL_ALARM_INST : Diag_Alarm;
      SUP_ALARM_INST : Diag_Alarm;
      STEP_TIME_ALARM_INST : Diag_Alarm;
      IEC_TIMER_INST : IEC_TIMER;
      TRANSACTION_FLAG : Bool := false;
   END_VAR
   VAR_TEMP
      txStartCondition : Bool;
      tdTckDiff : DInt;
      txReleaseConvIn : Bool;
   END_VAR
   VAR_TEMP   // added for the SCL form of the ladder/FBD networks
      _w1 : Bool;
   END_VAR
   // SINI[0] := 2;
   // LSTT[0] := 255;
   // LSTT[1] := 255;
   // LSTT[2] := 255;
   // LSTT[3] := 255;
   // LSTT[4] := 255;
   // LSTT[5] := 255;
   // LSTT[6] := 255;
   // LSTT[7] := 1;
   // ATAJ[1] := 1;
   // ATAJ[2] := 2;
   // ATAJ[3] := 6;
   // ATAJ[4] := 4;
   // ATAJ[5] := 5;
   // ATAJ[6] := 3;
   // ATAJ[7] := 7;
   // ATAB[0] := 4;
   // ATAB[1] := 1;
   // ATAB[2] := 2;
   // ATAB[3] := 3;
   // ATAB[5] := 5;
   // ATAB[6] := 6;
   // ATAB[7] := 7;
   // PSTT[1] := 1;
   // PSTT[2] := 2;
   // PSTT[3] := 3;
   // PSTT[5] := 4;
   // PSTT[6] := 5;
   // PSTT[7] := 6;
   // NSTT[0] := 1;
   // NSTT[1] := 2;
   // NSTT[2] := 7;
   // NSTT[3] := 6;
   // NSTT[4] := 4;
   // NSTT[5] := 8;
   // NSTT[6] := 6;
   // NSTT[7] := 1;
   // ASSJ[1] := 1;
   // ASSJ[2] := 2;
   // ASSJ[3] := 3;
   // ASSJ[4] := 4;
   // ASSJ[5] := 5;
   // ASSJ[6] := 6;
   // ASSB[1] := 1;
   // ASSB[2] := 2;
   // ASSB[3] := 3;
   // ASSB[4] := 4;
   // ASSB[5] := 5;
   // ASSB[6] := 6;
   // PTTS[0] := 255;
   // PTTS[2] := 1;
   // PTTS[3] := 13;
   // PTTS[4] := 4;
   // PTTS[5] := 14;
   // PTTS[6] := 3;
   // NTTS[1] := 1;
   // NTTS[2] := 2;
   // NTTS[3] := 3;
   // NTTS[4] := 5;
   // NTTS[5] := 6;
   // NTTS[6] := 7;
   // SW_SQTS[1] := 1;
   // SW_SQTS[2] := 1;
   // SW_SQTS[3] := 2;
   // SW_SQTS[4] := 3;
   // SW_SQTS[5] := 3;
   // SW_SQTS[6] := 4;
   // TVX[0] := 16#1;
   // TTX[0] := 16#1;
   // TSX[0] := 16#1;
   // S00X[0] := 16#1;
   // SOFFX[0] := 16#1;
   // SONX[0] := 16#1;
   // SAX[0] := 16#1;
   // SERRX[0] := 16#1;
   // SMX[0] := 16#1;
   // S0X[0] := 16#1;
   // S1X[0] := 16#1;
   // LSTT[8] := 255;
   // ATAJ[8] := 8;
   // ATAB[8] := 8;
   // PSTT[8] := 7;
   // NSTT[8] := 15;
   // ASSJ[7] := 7;
   // ASSB[7] := 7;
   // PTTS[7] := 2;
   // NTTS[7] := 8;
   // SW_SQTS[7] := 1;
   // LSTT[9] := 255;
   // LSTT[10] := 255;
   // LSTT[11] := 255;
   // ATAJ[9] := 9;
   // ATAJ[10] := 10;
   // ATAJ[11] := 11;
   // ATAB[9] := 9;
   // ATAB[10] := 10;
   // ATAB[11] := 11;
   // PSTT[9] := 8;
   // PSTT[10] := 9;
   // PSTT[11] := 10;
   // NSTT[9] := 13;
   // NSTT[10] := 11;
   // NSTT[11] := 16;
   // ASSJ[8] := 8;
   // ASSJ[9] := 9;
   // ASSJ[10] := 10;
   // ASSB[8] := 8;
   // ASSB[9] := 9;
   // ASSB[10] := 10;
   // PTTS[8] := 5;
   // PTTS[9] := 15;
   // PTTS[10] := 17;
   // NTTS[8] := 9;
   // NTTS[9] := 10;
   // NTTS[10] := 11;
   // SW_SQTS[8] := 3;
   // SW_SQTS[9] := 2;
   // SW_SQTS[10] := 1;
   // LSTT[12] := 255;
   // LSTT[13] := 255;
   // ATAJ[12] := 12;
   // ATAJ[13] := 13;
   // ATAB[12] := 12;
   // ATAB[13] := 13;
   // PSTT[12] := 11;
   // PSTT[13] := 12;
   // NSTT[12] := 17;
   // NSTT[13] := 3;
   // ASSJ[11] := 11;
   // ASSJ[12] := 12;
   // ASSB[11] := 11;
   // ASSB[12] := 12;
   // PTTS[11] := 10;
   // PTTS[12] := 19;
   // NTTS[11] := 12;
   // NTTS[12] := 13;
   // SW_SQTS[11] := 2;
   // SW_SQTS[12] := 2;
   // LSTT[14] := 255;
   // LSTT[15] := 255;
   // ATAJ[14] := 14;
   // ATAJ[15] := 15;
   // ATAB[14] := 14;
   // ATAB[15] := 16;
   // PSTT[14] := 13;
   // PSTT[15] := 14;
   // NSTT[14] := 5;
   // NSTT[15] := 9;
   // ASSJ[13] := 13;
   // ASSJ[14] := 14;
   // ASSB[13] := 13;
   // ASSB[14] := 14;
   // PTTS[13] := 9;
   // PTTS[14] := 18;
   // NTTS[13] := 14;
   // NTTS[14] := 15;
   // SW_SQTS[13] := 3;
   // SW_SQTS[14] := 1;
   // LSTT[16] := 16;
   // LSTT[17] := 255;
   // ATAJ[16] := 16;
   // ATAJ[17] := 17;
   // ATAB[16] := 15;
   // ATAB[17] := 17;
   // PSTT[16] := 14;
   // PSTT[17] := 15;
   // NSTT[16] := 16;
   // NSTT[17] := 10;
   // ASSJ[15] := 15;
   // ASSJ[16] := 16;
   // ASSB[15] := 15;
   // ASSB[16] := 16;
   // PTTS[15] := 8;
   // PTTS[16] := 11;
   // NTTS[15] := 17;
   // NTTS[16] := 18;
   // SW_SQTS[15] := 1;
   // SW_SQTS[16] := 1;
   // LSTT[18] := 255;
   // LSTT[19] := 255;
   // ATAJ[18] := 18;
   // ATAJ[19] := 19;
   // ATAB[18] := 18;
   // ATAB[19] := 19;
   // PSTT[18] := 16;
   // PSTT[19] := 17;
   // NSTT[18] := 14;
   // NSTT[19] := 12;
   // ASSJ[17] := 17;
   // ASSB[17] := 17;
   // PTTS[17] := 12;
   // NTTS[17] := 19;
   // SW_SQTS[17] := 2;
BEGIN
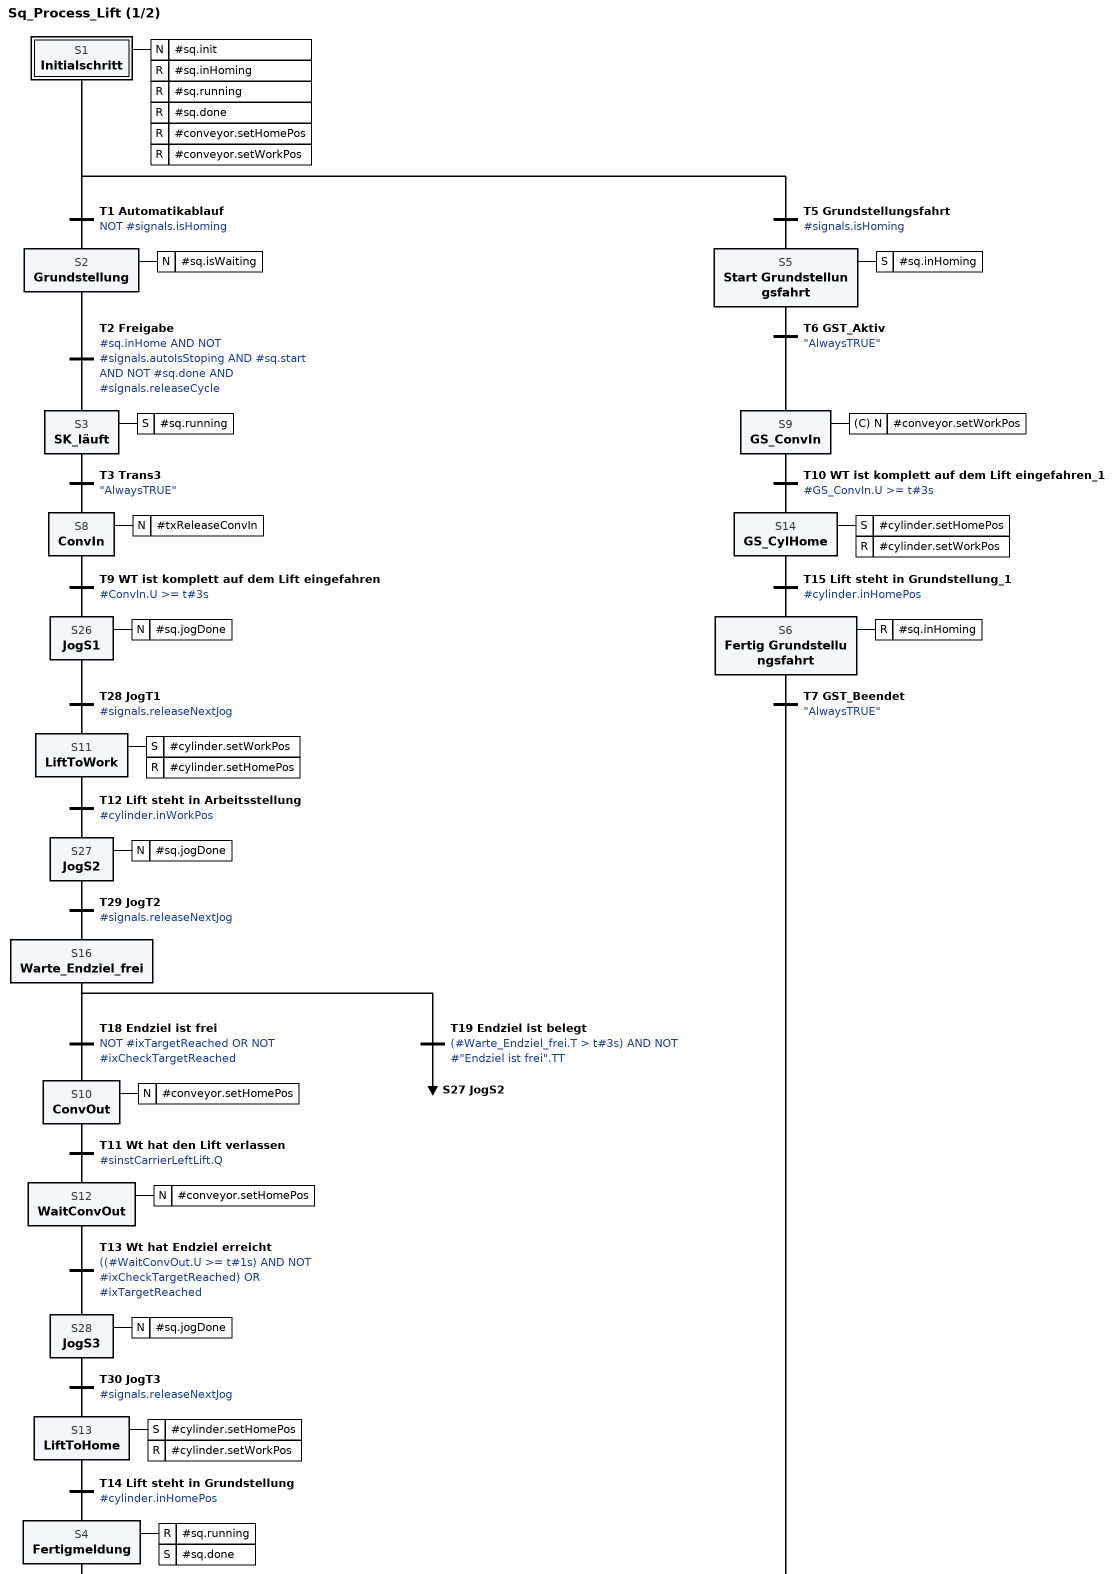
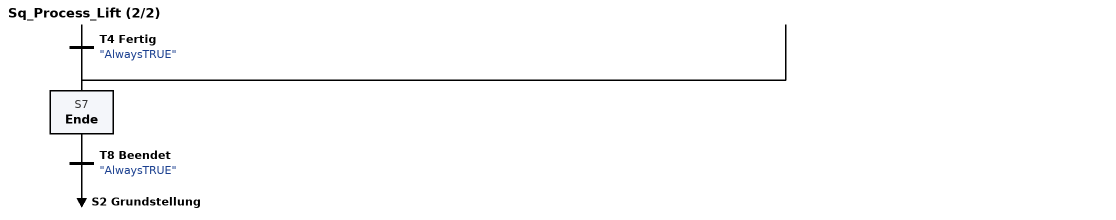
   // permanent pre-instructions
   NETWORK 1
   TITLE = Schrittkette verfügbar
      #sq.exists := true;
   NETWORK 2
   TITLE = WT auf dem Lift
      #sinstCarrierOnLift(IN := #ixCarrierPresent, PT := #itCarrierReactionDelay);   // TON
   NETWORK 3
   TITLE = WT hat Lift verlassen
      #sinstCarrierLeftLift(IN := NOT #ixCarrierPresent, PT := #itCarrierReactionDelay);   // TON
   NETWORK 4
   TITLE = Schrittkette in Grundstellung (Erweiterbar)
      #sq.inHome := #Grundstellung.X AND #cylinder.inHomePos AND NOT #ixExternReqConvIn;
   NETWORK 5
   TITLE = Startbedingung (Erweiterbar)
      #txStartCondition := #ixStart AND #sinstCarrierOnLift.Q;
   NETWORK 6
   TITLE = Schrittkette starten
      #sq.start := NOT #sq.running AND #signals.releaseCycle AND NOT #signals.isHoming AND #txStartCondition;
      IF #sq.start THEN #sq.done := FALSE; END_IF;
   NETWORK 7
   TITLE = ReleaseCycle Timer
      // ENO of a box is taken as its EN; it also drops when the box reports an error
      #_w1 := NOT #ERR_FLT AND #sstReleaseCycle.ErrorAck;   // falling edge
      #sstReleaseCycle.ErrorAck := #ERR_FLT;
      IF (#S_NO <> #sstReleaseCycle.No_LastCycle) OR #_w1 THEN
          #sstReleaseCycle.T := T#0MS;
          #sstReleaseCycle.TckPrev := #sstReleaseCycle.Tck;
          #sstReleaseCycle.No_LastCycle := #S_NO;
      END_IF;
      #sstReleaseCycle.Tck := TIME_TCK();
      #tdTckDiff := #sstReleaseCycle.Tck - #sstReleaseCycle.TckPrev;
      #sstReleaseCycle.TckPrev := #sstReleaseCycle.Tck;
      IF (0 <= #tdTckDiff) AND (#tdTckDiff <= 1000) AND #signals.releaseCycle THEN
          #sstReleaseCycle.T := #sstReleaseCycle.T + #tdTckDiff;
      END_IF;

   // sequencer 1
   INITIAL_STEP Initialschritt:   // S1, max time T#10S, warning time T#7S
              N    #sq.init
              R    #sq.inHoming
              R    #sq.running
              R    #sq.done
              R    #conveyor.setHomePos
              R    #conveyor.setWorkPos
   END_STEP
   TRANSITION Automatikablauf FROM Initialschritt TO Grundstellung   // T1
      := NOT #signals.isHoming;
   END_TRANSITION
   TRANSITION Grundstellungsfahrt FROM Initialschritt TO "Start Grundstellungsfahrt"   // T5
      := #signals.isHoming;
   END_TRANSITION
   STEP Grundstellung:   // S2, max time T#10S, warning time T#7S
              N    #sq.isWaiting
   END_STEP
   TRANSITION Freigabe FROM Grundstellung TO SK_läuft   // T2
      := #sq.inHome AND NOT #signals.autoIsStoping AND #sq.start AND NOT #sq.done AND #signals.releaseCycle;
   END_TRANSITION
   STEP SK_läuft:   // S3, max time T#10S, warning time T#7S
              S    #sq.running
   END_STEP
   TRANSITION Trans3 FROM SK_läuft TO ConvIn   // T3
      := "AlwaysTRUE";
   END_TRANSITION
   STEP Fertigmeldung:   // S4, max time T#10S, warning time T#7S
              R    #sq.running
              S    #sq.done
   END_STEP
   TRANSITION Fertig FROM Fertigmeldung TO Ende   // T4
      := "AlwaysTRUE";
   END_TRANSITION
   STEP "Start Grundstellungsfahrt":   // S5, max time T#10S, warning time T#7S
              S    #sq.inHoming
   END_STEP
   TRANSITION GST_Aktiv FROM "Start Grundstellungsfahrt" TO GS_ConvIn   // T6
      := "AlwaysTRUE";
   END_TRANSITION
   STEP "Fertig Grundstellungsfahrt":   // S6, max time T#10S, warning time T#7S
              R    #sq.inHoming
   END_STEP
   TRANSITION GST_Beendet FROM "Fertig Grundstellungsfahrt" TO Ende   // T7
      := "AlwaysTRUE";
   END_TRANSITION
   STEP Ende:   // S7, max time T#10S, warning time T#7S
   END_STEP
   TRANSITION Beendet FROM Ende TO Grundstellung   // T8, jump
      := "AlwaysTRUE";
   END_TRANSITION
   STEP ConvIn:   // S8, max time T#10S, warning time T#7S
      supervision V := (#sstReleaseCycle.T >= #itMaxRuntime) OR (#ConvIn.X AND #conveyor.inError);
      // WT soll komplett einfahren
              N    #txReleaseConvIn
   END_STEP
   TRANSITION "WT ist komplett auf dem Lift eingefahren" FROM ConvIn TO JogS1   // T9
      := #ConvIn.U >= t#3s;
   END_TRANSITION
   STEP JogS1:   // S26, max time T#10S, warning time T#7S
              N    #sq.jogDone
   END_STEP
   TRANSITION JogT1 FROM JogS1 TO LiftToWork   // T28
      := #signals.releaseNextJog;
   END_TRANSITION
   STEP ConvOut:   // S10, max time T#10S, warning time T#7S
      supervision V := (#sstReleaseCycle.T >= #itMaxRuntime) OR (#ConvOut.X AND #conveyor.inError);
              N    #conveyor.setHomePos
   END_STEP
   TRANSITION "Wt hat den Lift verlassen" FROM ConvOut TO WaitConvOut   // T11
      := #sinstCarrierLeftLift.Q;
   END_TRANSITION
   STEP LiftToWork:   // S11, max time T#10S, warning time T#7S
      supervision V := (#sstReleaseCycle.T >= #itMaxRuntime) OR (#LiftToWork.X AND #cylinder.inError);
              S    #cylinder.setWorkPos
              R    #cylinder.setHomePos
   END_STEP
   TRANSITION "Lift steht in Arbeitsstellung" FROM LiftToWork TO JogS2   // T12
      := #cylinder.inWorkPos;
   END_TRANSITION
   STEP JogS2:   // S27, max time T#10S, warning time T#7S
              N    #sq.jogDone
   END_STEP
   TRANSITION JogT2 FROM JogS2 TO Warte_Endziel_frei   // T29
      := #signals.releaseNextJog;
   END_TRANSITION
   STEP WaitConvOut:   // S12, max time T#10S, warning time T#7S
      supervision V := (#sstReleaseCycle.T >= #itMaxRuntime) OR (#WaitConvOut.X AND #conveyor.inError);
              N    #conveyor.setHomePos
   END_STEP
   TRANSITION "Wt hat Endziel erreicht" FROM WaitConvOut TO JogS3   // T13
      := ((#WaitConvOut.U >= t#1s) AND NOT #ixCheckTargetReached) OR #ixTargetReached;
   END_TRANSITION
   STEP JogS3:   // S28, max time T#10S, warning time T#7S
              N    #sq.jogDone
   END_STEP
   TRANSITION JogT3 FROM JogS3 TO LiftToHome   // T30
      := #signals.releaseNextJog;
   END_TRANSITION
   STEP LiftToHome:   // S13, max time T#10S, warning time T#7S
      supervision V := (#sstReleaseCycle.T >= #itMaxRuntime) OR (#LiftToHome.X AND #cylinder.inError);
              S    #cylinder.setHomePos
              R    #cylinder.setWorkPos
   END_STEP
   TRANSITION "Lift steht in Grundstellung" FROM LiftToHome TO Fertigmeldung   // T14
      := #cylinder.inHomePos;
   END_TRANSITION
   STEP GS_ConvIn:   // S9, max time T#10S, warning time T#7S
      interlock C := NOT #GS_ConvIn.VA OR NOT #signals.isInError;
      supervision V := (#sstReleaseCycle.T >= #itMaxRuntime) OR (#GS_ConvIn.X AND #conveyor.inError);
      // WT soll komplett einfahren
      (C)     N    #conveyor.setWorkPos
   END_STEP
   TRANSITION "WT ist komplett auf dem Lift eingefahren_1" FROM GS_ConvIn TO GS_CylHome   // T10
      := #GS_ConvIn.U >= t#3s;
   END_TRANSITION
   STEP GS_CylHome:   // S14, max time T#10S, warning time T#7S
      supervision V := (#sstReleaseCycle.T >= #itMaxRuntime) OR (#GS_CylHome.X AND #cylinder.inError);
              S    #cylinder.setHomePos
              R    #cylinder.setWorkPos
   END_STEP
   TRANSITION "Lift steht in Grundstellung_1" FROM GS_CylHome TO "Fertig Grundstellungsfahrt"   // T15
      := #cylinder.inHomePos;
   END_TRANSITION
   STEP Warte_Endziel_frei:   // S16, max time T#10S, warning time T#7S
   END_STEP
   TRANSITION "Endziel ist frei" FROM Warte_Endziel_frei TO ConvOut   // T18
      := NOT #ixTargetReached OR NOT #ixCheckTargetReached;
   END_TRANSITION
   TRANSITION "Endziel ist belegt" FROM Warte_Endziel_frei TO JogS2   // T19, jump
      := (#Warte_Endziel_frei.T > t#3s) AND NOT #"Endziel ist frei".TT;
   END_TRANSITION

   // permanent post-instructions
   NETWORK 1
   TITLE = Störungssignal weitergeben
      #sq.error := #ERR_FLT;
   NETWORK 2
   TITLE = Ablauf ist aktiv
      #qxIsActive := #sq.running;
   NETWORK 3
   TITLE = steht in Grundstellung
      #qxIsInHome := #sq.inHome AND NOT #sq.running;
   NETWORK 4
   TITLE = Förderband Einlauf in Lift einschalten
      #conveyor.setWorkPos := ((#ixExternReqConvIn AND NOT #qxIsActive) OR #txReleaseConvIn) AND #signals.releaseCycle;
END_FUNCTION_BLOCK

FUNCTION_BLOCK "Sq_Process_IndexingUnit"   // FB9304, GRAPH_PLUS
{ S7_Optimized_Access := 'TRUE' }
VERSION : 0.1
   VAR_INPUT
      OFF_SQ : Bool := false;   // Kette ausschalten
      INIT_SQ : Bool := false;   // Kette in Initialzustand versetzen
      ACK_EF : Bool := false;   // Alle Fehler und Störungen quittieren
      S_PREV : Bool := false;   // Vorherigen Schritt am Parameter S_NO ausgeben
      S_NEXT : Bool := false;   // Nächsten Schritt am Parameter S_NO anzeigen
      SW_AUTO : Bool := false;   // Automatischer Betrieb
      SW_TAP : Bool := false;   // Halbautomatisch/Weiterschalten mit Transition
      SW_TOP : Bool := false;   // Halbautomatisch/Ignoriere Transition
      SW_MAN : Bool := false;   // Handbetrieb
      S_SEL : Int := 0;   // Schritt auswählen, der an S_NO ausgegeben werden soll
      S_ON : Bool := false;   // Schritt aktivieren, der an Parameter S_NO anliegt
      S_OFF : Bool := false;   // Schritt deaktivieren, der an Parameter S_NO anliegt
      T_PUSH : Bool := false;   // Schaltfreigabe für Transition im halbautomatischen Betrieb
      ixStart : Bool := true;   // Startfreigabe
      ixCarrierPresent : Bool;   // WT auf dem Indexer vorhanden
      ixCheckTargetReached : Bool := false;   // 0 = Keine Sensor-Zielüberwachung nach Lift vorhanden
      ixTargetReached : Bool := false;   // WT-Sensor des nächsten Ziels
      ixReleaseHoming : Bool := true;   // Freigabe Grundstellungsfahrt
      ixReleaseTransfer : Bool := true;   // Freigabe der nächsten Position um WT weiterzutakten
      itCarrierReactionDelay : Time := T#350ms;   // Verzögerungszeit für die WT-Erkennung
      itMaxRuntime : Time := t#10s;   // Maximale Laufzeit für diesen Prozess
   END_VAR
   VAR_OUTPUT
      S_NO : Int := 0;   // Schrittnummer
      S_MORE : Bool := false;   // Weitere Schritte sind vorhanden und können in S_NO angezeigt werden.
      S_ACTIVE : Bool := false;   // Schritt, der an Parameter S_NO angezeigt wird, ist aktiv
      ERR_FLT : Bool := false;   // Sammelfehler Interlock oder Supervision
      AUTO_ON : Bool := false;   // Automatischer Betrieb eingeschaltet
      TAP_ON : Bool := false;   // Halbautomatischer Betrieb/Schritt mit Transition eingeschaltet
      TOP_ON : Bool := false;   // Halbautomatischer Betrieb/Ignoriere Transition eingeschaltet
      MAN_ON : Bool := false;   // Handbetrieb eingeschaltet
      qxIsActive : Bool;   // Schrittkette läuft
      qxIsInHome : Bool;   // steht in Grundstellung
      qxCarrierIsDone : Bool;   // WT-Träger ist fertig bearbeitet worden
   END_VAR
   VAR_IN_OUT
      signals : "typeStationSignals";   // Stationssteuersignale
      sq : "typeStepSequence";   // Schrittkettensteuersignale
      cylinder_lift : "typeActor_2Out2In";   // Aktor des Heber
      cylinder_stopper : "typeActor_1Out1In";   // Aktor für den Stopper
      releaseWorkStep : Bool;   // Freigabe für den externen Arbeitsschritt (muss extern zurückgesetzt werden)
   END_VAR
   VAR
      sstReleaseCycle : Struct
         ErrorAck : Bool;
         No_LastCycle : Int;
         T : Time;   // Aktive Zeit des ReleaseCycle
         Tck : Time;
         TckPrev : Time;
      END_STRUCT;
      sinstCarrierOnIndexer : TON_TIME;
      sinstCarrierLeftIndexer : TON_TIME;
      HMI_INFO : Array[0..8] of UInt;
      IF_PAR : G7_IfParPlus_V6;
      RT_DATA : G7_RTDataPlus_V6;   // Interner Datenbereich
      Automatikablauf : G7_TransitionPlus_V6;   // Transitionsstruktur
      Freigabe : G7_TransitionPlus_V6;   // Transitionsstruktur
      Trans3 : G7_TransitionPlus_V6;   // Transitionsstruktur
      Fertig : G7_TransitionPlus_V6;   // Transitionsstruktur
      Grundstellungsfahrt : G7_TransitionPlus_V6;   // Transitionsstruktur
      GST_Aktiv : G7_TransitionPlus_V6;   // Transitionsstruktur
      GST_Beendet : G7_TransitionPlus_V6;   // Transitionsstruktur
      Beendet : G7_TransitionPlus_V6;   // Transitionsstruktur
      TargetIsReached : G7_TransitionPlus_V6;   // Transitionsstruktur / Transition structure
      "Lift steht in Grundstellung_1" : G7_TransitionPlus_V6;   // Transitionsstruktur / Transition structure
      "Lift steht in Arbeitsstellung_1" : G7_TransitionPlus_V6;   // Transitionsstruktur / Transition structure
      "Lift steht in Arbeitsstellung_2" : G7_TransitionPlus_V6;   // Transitionsstruktur / Transition structure
      "WT hat Stopper verlassen" : G7_TransitionPlus_V6;   // Transitionsstruktur / Transition structure
      CarrierIsNotDone : G7_TransitionPlus_V6;   // Transitionsstruktur / Transition structure
      CarrierIsDone : G7_TransitionPlus_V6;   // Transitionsstruktur / Transition structure
      WorkstepDone : G7_TransitionPlus_V6;   // Transitionsstruktur / Transition structure
      NotDone : G7_TransitionPlus_V6;   // Transitionsstruktur / Transition structure
      WorkstepIsReleased : G7_TransitionPlus_V6;   // Transitionsstruktur / Transition structure
      EndzielFrei : G7_TransitionPlus_V6;   // Transitionsstruktur / Transition structure
      EndzielNichtFrei : G7_TransitionPlus_V6;   // Transitionsstruktur / Transition structure
      JogT1 : G7_TransitionPlus_V6;   // Transitionsstruktur / Transition structure
      JogT2 : G7_TransitionPlus_V6;   // Transitionsstruktur / Transition structure
      Initialschritt : G7_StepPlus_V6;   // Schrittstruktur
      Grundstellung : G7_StepPlus_V6;   // Schrittstruktur
      SK_läuft : G7_StepPlus_V6;   // Schrittstruktur
      Fertigmeldung : G7_StepPlus_V6;   // Schrittstruktur
      "Start Grundstellungsfahrt" : G7_StepPlus_V6;   // Schrittstruktur
      "Fertig Grundstellungsfahrt" : G7_StepPlus_V6;   // Schrittstruktur
      Ende : G7_StepPlus_V6;   // Schrittstruktur
      WaitForTarget : G7_StepPlus_V6;   // Schrittstruktur / Step structure
      GS_CylHome : G7_StepPlus_V6;   // Schrittstruktur / Step structure
      IndexerWorkPos : G7_StepPlus_V6;   // Schrittstruktur / Step structure
      IndexerHomePos : G7_StepPlus_V6;   // Schrittstruktur / Step structure
      OpenStopper : G7_StepPlus_V6;   // Schrittstruktur / Step structure
      Decision : G7_StepPlus_V6;   // Schrittstruktur / Step structure
      CheckWorkstepDone : G7_StepPlus_V6;   // Schrittstruktur / Step structure
      Release : G7_StepPlus_V6;   // Schrittstruktur / Step structure
      Warte_Endziel_frei : G7_StepPlus_V6;   // Schrittstruktur / Step structure
      JogS1 : G7_StepPlus_V6;   // Schrittstruktur / Step structure
      JogS2 : G7_StepPlus_V6;   // Schrittstruktur / Step structure
      SINI : Array[0..1] of USInt;
      LSTT : Array[0..21] of USInt;
      ATAJ : Array[0..21] of USInt;
      ATAB : Array[0..21] of USInt;
      PSTT : Array[0..21] of USInt;
      NSTT : Array[0..21] of USInt;
      ASSJ : Array[0..17] of USInt;
      ASSB : Array[0..17] of USInt;
      PTTS : Array[0..17] of USInt;
      NTTS : Array[0..17] of USInt;
      SW_SQTS : Array[0..17] of USInt;
      SWITCH : Array[0..7] of USInt;
      TVX : Array[0..9] of USInt;
      TTX : Array[0..9] of USInt;
      TSX : Array[0..1] of USInt;
      S00X : Array[0..1] of USInt;
      SOFFX : Array[0..1] of USInt;
      SONX : Array[0..1] of USInt;
      SAX : Array[0..1] of USInt;
      SERRX : Array[0..18] of USInt;
      SMX : Array[0..18] of USInt;
      S0X : Array[0..18] of USInt;
      S1X : Array[0..18] of USInt;
      IL_ALARM_INST : Diag_Alarm;
      SUP_ALARM_INST : Diag_Alarm;
      STEP_TIME_ALARM_INST : Diag_Alarm;
      IEC_TIMER_INST : IEC_TIMER;
      TRANSACTION_FLAG : Bool := false;
   END_VAR
   VAR_TEMP
      txStartCondition : Bool;
      tdTckDiff : DInt;
      txCheckWorkStep : Bool;
   END_VAR
   VAR_TEMP   // added for the SCL form of the ladder/FBD networks
      _w1 : Bool;
   END_VAR
   // SINI[0] := 2;
   // LSTT[0] := 255;
   // LSTT[1] := 255;
   // LSTT[2] := 255;
   // LSTT[3] := 255;
   // LSTT[4] := 255;
   // LSTT[5] := 255;
   // LSTT[6] := 255;
   // LSTT[7] := 1;
   // ATAJ[1] := 1;
   // ATAJ[2] := 2;
   // ATAJ[3] := 6;
   // ATAJ[4] := 4;
   // ATAJ[5] := 5;
   // ATAJ[6] := 3;
   // ATAJ[7] := 7;
   // ATAB[0] := 4;
   // ATAB[1] := 1;
   // ATAB[2] := 2;
   // ATAB[3] := 3;
   // ATAB[5] := 5;
   // ATAB[6] := 6;
   // ATAB[7] := 7;
   // PSTT[1] := 1;
   // PSTT[2] := 2;
   // PSTT[3] := 3;
   // PSTT[5] := 4;
   // PSTT[6] := 5;
   // PSTT[7] := 6;
   // NSTT[0] := 1;
   // NSTT[1] := 2;
   // NSTT[2] := 12;
   // NSTT[3] := 6;
   // NSTT[4] := 4;
   // NSTT[5] := 8;
   // NSTT[6] := 6;
   // NSTT[7] := 1;
   // ASSJ[1] := 1;
   // ASSJ[2] := 2;
   // ASSJ[3] := 3;
   // ASSJ[4] := 4;
   // ASSJ[5] := 5;
   // ASSJ[6] := 6;
   // ASSB[1] := 1;
   // ASSB[2] := 2;
   // ASSB[3] := 3;
   // ASSB[4] := 4;
   // ASSB[5] := 5;
   // ASSB[6] := 6;
   // PTTS[0] := 255;
   // PTTS[2] := 1;
   // PTTS[3] := 8;
   // PTTS[4] := 4;
   // PTTS[5] := 9;
   // PTTS[6] := 3;
   // NTTS[1] := 1;
   // NTTS[2] := 2;
   // NTTS[3] := 3;
   // NTTS[4] := 5;
   // NTTS[5] := 6;
   // NTTS[6] := 7;
   // SW_SQTS[1] := 1;
   // SW_SQTS[2] := 1;
   // SW_SQTS[3] := 2;
   // SW_SQTS[4] := 3;
   // SW_SQTS[5] := 3;
   // SW_SQTS[6] := 4;
   // TVX[0] := 16#1;
   // TTX[0] := 16#1;
   // TSX[0] := 16#1;
   // S00X[0] := 16#1;
   // SOFFX[0] := 16#1;
   // SONX[0] := 16#1;
   // SAX[0] := 16#1;
   // SERRX[0] := 16#1;
   // SMX[0] := 16#1;
   // S0X[0] := 16#1;
   // S1X[0] := 16#1;
   // LSTT[8] := 255;
   // ATAJ[8] := 8;
   // ATAB[8] := 8;
   // PSTT[8] := 7;
   // NSTT[8] := 3;
   // ASSJ[7] := 7;
   // ASSB[7] := 7;
   // PTTS[7] := 12;
   // NTTS[7] := 8;
   // SW_SQTS[7] := 2;
   // LSTT[9] := 255;
   // LSTT[10] := 255;
   // LSTT[11] := 255;
   // ATAJ[9] := 9;
   // ATAJ[10] := 10;
   // ATAJ[11] := 14;
   // ATAB[9] := 9;
   // ATAB[10] := 10;
   // ATAB[11] := 11;
   // PSTT[9] := 8;
   // PSTT[10] := 9;
   // PSTT[11] := 10;
   // NSTT[9] := 5;
   // NSTT[10] := 14;
   // NSTT[11] := 17;
   // ASSJ[8] := 8;
   // ASSJ[9] := 9;
   // ASSJ[10] := 10;
   // ASSB[8] := 8;
   // ASSB[9] := 9;
   // ASSB[10] := 10;
   // PTTS[8] := 5;
   // PTTS[9] := 13;
   // PTTS[10] := 15;
   // NTTS[8] := 9;
   // NTTS[9] := 10;
   // NTTS[10] := 11;
   // SW_SQTS[8] := 3;
   // SW_SQTS[9] := 5;
   // SW_SQTS[10] := 6;
   // LSTT[12] := 255;
   // LSTT[13] := 255;
   // ATAJ[12] := 12;
   // ATAJ[13] := 13;
   // ATAB[12] := 12;
   // ATAB[13] := 14;
   // PSTT[12] := 11;
   // PSTT[13] := 12;
   // NSTT[12] := 7;
   // NSTT[13] := 9;
   // ASSJ[11] := 11;
   // ASSJ[12] := 12;
   // ASSB[11] := 11;
   // ASSB[12] := 12;
   // PTTS[11] := 18;
   // PTTS[12] := 2;
   // NTTS[11] := 12;
   // NTTS[12] := 13;
   // SW_SQTS[11] := 2;
   // SW_SQTS[12] := 1;
   // LSTT[14] := 255;
   // LSTT[15] := 255;
   // ATAJ[14] := 11;
   // ATAJ[15] := 15;
   // ATAB[14] := 13;
   // ATAB[15] := 16;
   // PSTT[14] := 12;
   // PSTT[15] := 13;
   // NSTT[14] := 17;
   // NSTT[15] := 10;
   // ASSJ[13] := 13;
   // ASSJ[14] := 14;
   // ASSB[13] := 13;
   // ASSB[14] := 14;
   // PTTS[13] := 20;
   // PTTS[14] := 10;
   // NTTS[13] := 15;
   // NTTS[14] := 17;
   // SW_SQTS[13] := 5;
   // SW_SQTS[14] := 5;
   // LSTT[16] := 16;
   // ATAJ[16] := 16;
   // ATAB[16] := 15;
   // PSTT[16] := 13;
   // NSTT[16] := 16;
   // LSTT[17] := 255;
   // LSTT[18] := 255;
   // ATAJ[17] := 17;
   // ATAJ[18] := 18;
   // ATAB[17] := 17;
   // ATAB[18] := 19;
   // PSTT[17] := 14;
   // PSTT[18] := 15;
   // NSTT[17] := 16;
   // NSTT[18] := 11;
   // ASSJ[15] := 15;
   // ASSB[15] := 15;
   // PTTS[15] := 21;
   // NTTS[15] := 18;
   // SW_SQTS[15] := 7;
   // LSTT[19] := 17;
   // ATAJ[19] := 19;
   // ATAB[19] := 18;
   // PSTT[19] := 15;
   // NSTT[19] := 17;
   // ASSJ[16] := 16;
   // ASSB[16] := 16;
   // PTTS[16] := 17;
   // NTTS[16] := 20;
   // SW_SQTS[16] := 5;
   // LSTT[20] := 255;
   // LSTT[21] := 255;
   // ATAJ[20] := 20;
   // ATAJ[21] := 21;
   // ATAB[20] := 20;
   // ATAB[21] := 21;
   // PSTT[20] := 16;
   // PSTT[21] := 17;
   // NSTT[20] := 13;
   // NSTT[21] := 15;
   // ASSJ[17] := 17;
   // ASSB[17] := 17;
   // PTTS[17] := 11;
   // NTTS[17] := 21;
   // SW_SQTS[17] := 7;
BEGIN
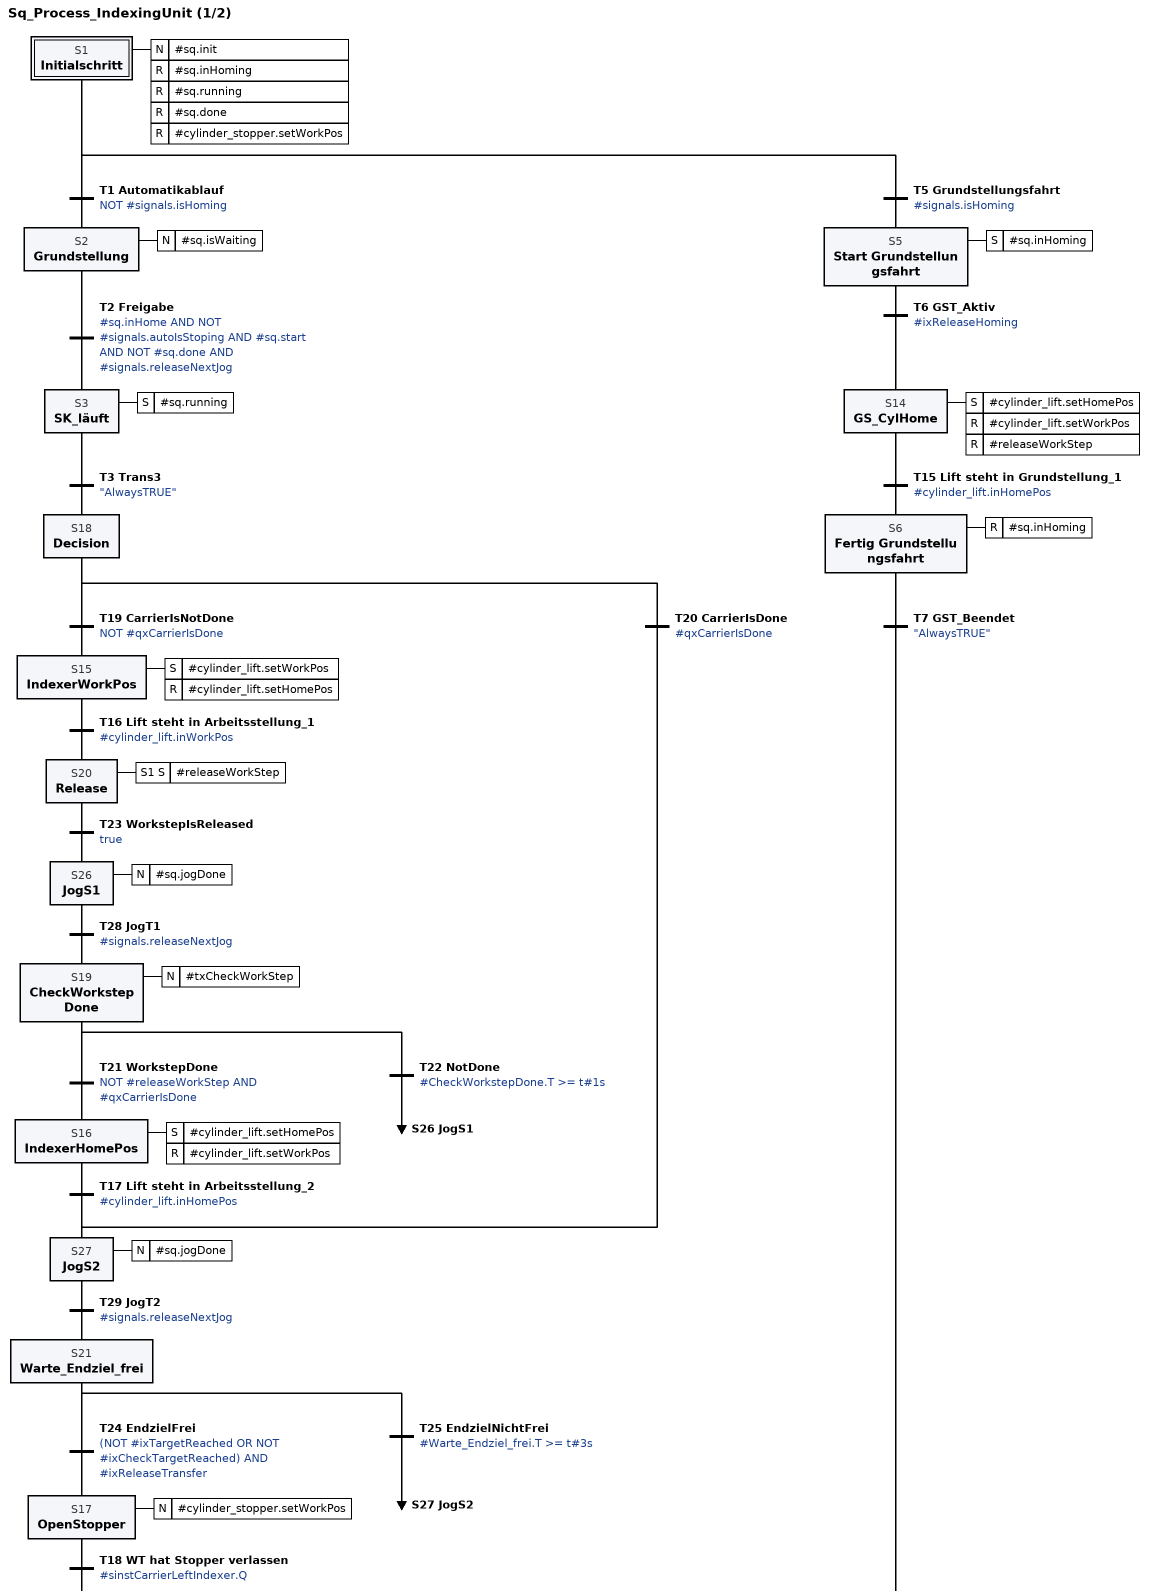
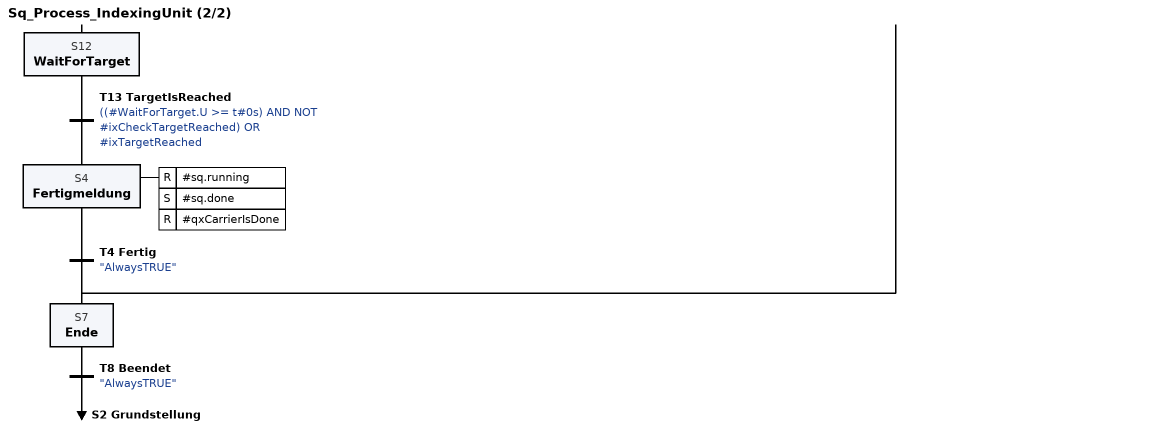
   // permanent pre-instructions
   NETWORK 1
   TITLE = Schrittkette verfügbar
      #sq.exists := true;
   NETWORK 2
   TITLE = WT auf dem Indexer
      #sinstCarrierOnIndexer(IN := #ixCarrierPresent, PT := #itCarrierReactionDelay);   // TON
   NETWORK 3
   TITLE = WT hat den Indexer verlassen
      #sinstCarrierLeftIndexer(IN := NOT #ixCarrierPresent, PT := #itCarrierReactionDelay);   // TON
   NETWORK 4
   TITLE = Schrittkette in Grundstellung (Erweitern)
      #sq.inHome := #Grundstellung.X AND #cylinder_lift.inHomePos AND #cylinder_stopper.inHomePos;
   NETWORK 5
   TITLE = Startbedingung (Erweitern)
      #txStartCondition := #ixStart AND #sinstCarrierOnIndexer.Q;
   NETWORK 6
   TITLE = Schrittkette starten
      #sq.start := #sq.inHome AND NOT #sq.running AND #signals.releaseCycle AND NOT #signals.isHoming AND #txStartCondition;
      IF #sq.start THEN #sq.done := FALSE; END_IF;
   NETWORK 7
   TITLE = ReleaseCycle Timer
      // ENO of a box is taken as its EN; it also drops when the box reports an error
      #_w1 := NOT #ERR_FLT AND #sstReleaseCycle.ErrorAck;   // falling edge
      #sstReleaseCycle.ErrorAck := #ERR_FLT;
      IF (#S_NO <> #sstReleaseCycle.No_LastCycle) OR #_w1 THEN
          #sstReleaseCycle.T := T#0MS;
          #sstReleaseCycle.TckPrev := #sstReleaseCycle.Tck;
          #sstReleaseCycle.No_LastCycle := #S_NO;
      END_IF;
      #sstReleaseCycle.Tck := TIME_TCK();
      #tdTckDiff := #sstReleaseCycle.Tck - #sstReleaseCycle.TckPrev;
      #sstReleaseCycle.TckPrev := #sstReleaseCycle.Tck;
      IF (0 <= #tdTckDiff) AND (#tdTckDiff <= 1000) AND #signals.releaseCycle THEN
          #sstReleaseCycle.T := #sstReleaseCycle.T + #tdTckDiff;
      END_IF;

   // sequencer 1
   INITIAL_STEP Initialschritt:   // S1, max time T#10S, warning time T#7S
              N    #sq.init
              R    #sq.inHoming
              R    #sq.running
              R    #sq.done
              R    #cylinder_stopper.setWorkPos
   END_STEP
   TRANSITION Automatikablauf FROM Initialschritt TO Grundstellung   // T1
      := NOT #signals.isHoming;
   END_TRANSITION
   TRANSITION Grundstellungsfahrt FROM Initialschritt TO "Start Grundstellungsfahrt"   // T5
      := #signals.isHoming;
   END_TRANSITION
   STEP Grundstellung:   // S2, max time T#10S, warning time T#7S
              N    #sq.isWaiting
   END_STEP
   TRANSITION Freigabe FROM Grundstellung TO SK_läuft   // T2
      := #sq.inHome AND NOT #signals.autoIsStoping AND #sq.start AND NOT #sq.done AND #signals.releaseNextJog;
   END_TRANSITION
   STEP SK_läuft:   // S3, max time T#10S, warning time T#7S
              S    #sq.running
   END_STEP
   TRANSITION Trans3 FROM SK_läuft TO Decision   // T3
      := "AlwaysTRUE";
   END_TRANSITION
   STEP Fertigmeldung:   // S4, max time T#10S, warning time T#7S
              R    #sq.running
              S    #sq.done
              R    #qxCarrierIsDone
   END_STEP
   TRANSITION Fertig FROM Fertigmeldung TO Ende   // T4
      := "AlwaysTRUE";
   END_TRANSITION
   STEP "Start Grundstellungsfahrt":   // S5, max time T#10S, warning time T#7S
              S    #sq.inHoming
   END_STEP
   TRANSITION GST_Aktiv FROM "Start Grundstellungsfahrt" TO GS_CylHome   // T6
      := #ixReleaseHoming;
   END_TRANSITION
   STEP "Fertig Grundstellungsfahrt":   // S6, max time T#10S, warning time T#7S
              R    #sq.inHoming
   END_STEP
   TRANSITION GST_Beendet FROM "Fertig Grundstellungsfahrt" TO Ende   // T7
      := "AlwaysTRUE";
   END_TRANSITION
   STEP Ende:   // S7, max time T#10S, warning time T#7S
   END_STEP
   TRANSITION Beendet FROM Ende TO Grundstellung   // T8, jump
      := "AlwaysTRUE";
   END_TRANSITION
   STEP JogS1:   // S26, max time T#10S, warning time T#7S
              N    #sq.jogDone
   END_STEP
   TRANSITION JogT1 FROM JogS1 TO CheckWorkstepDone   // T28
      := #signals.releaseNextJog;
   END_TRANSITION
   STEP IndexerHomePos:   // S16, max time T#10S, warning time T#7S
      supervision V := #IndexerHomePos.X AND #cylinder_lift.inError;
              S    #cylinder_lift.setHomePos
              R    #cylinder_lift.setWorkPos
   END_STEP
   TRANSITION "Lift steht in Arbeitsstellung_2" FROM IndexerHomePos TO JogS2   // T17
      := #cylinder_lift.inHomePos;
   END_TRANSITION
   STEP OpenStopper:   // S17, max time T#10S, warning time T#7S
      supervision V := #OpenStopper.X AND #cylinder_stopper.inError;
              N    #cylinder_stopper.setWorkPos
   END_STEP
   TRANSITION "WT hat Stopper verlassen" FROM OpenStopper TO WaitForTarget   // T18
      := #sinstCarrierLeftIndexer.Q;
   END_TRANSITION
   STEP JogS2:   // S27, max time T#10S, warning time T#7S
              N    #sq.jogDone
   END_STEP
   TRANSITION JogT2 FROM JogS2 TO Warte_Endziel_frei   // T29
      := #signals.releaseNextJog;
   END_TRANSITION
   STEP WaitForTarget:   // S12, max time T#10S, warning time T#7S
      supervision V := #sstReleaseCycle.T >= #itMaxRuntime;
   END_STEP
   TRANSITION TargetIsReached FROM WaitForTarget TO Fertigmeldung   // T13
      := ((#WaitForTarget.U >= t#0s) AND NOT #ixCheckTargetReached) OR #ixTargetReached;
   END_TRANSITION
   STEP Decision:   // S18, max time T#10S, warning time T#7S
   END_STEP
   TRANSITION CarrierIsNotDone FROM Decision TO IndexerWorkPos   // T19
      := NOT #qxCarrierIsDone;
   END_TRANSITION
   TRANSITION CarrierIsDone FROM Decision TO JogS2   // T20
      := #qxCarrierIsDone;
   END_TRANSITION
   STEP GS_CylHome:   // S14, max time T#10S, warning time T#7S
      supervision V := #GS_CylHome.X AND #cylinder_lift.inError;
              S    #cylinder_lift.setHomePos
              R    #cylinder_lift.setWorkPos
              R    #releaseWorkStep
   END_STEP
   TRANSITION "Lift steht in Grundstellung_1" FROM GS_CylHome TO "Fertig Grundstellungsfahrt"   // T15
      := #cylinder_lift.inHomePos;
   END_TRANSITION
   STEP IndexerWorkPos:   // S15, max time T#10S, warning time T#7S
      supervision V := #IndexerWorkPos.X AND #cylinder_lift.inError;
              S    #cylinder_lift.setWorkPos
              R    #cylinder_lift.setHomePos
   END_STEP
   TRANSITION "Lift steht in Arbeitsstellung_1" FROM IndexerWorkPos TO Release   // T16
      := #cylinder_lift.inWorkPos;
   END_TRANSITION
   STEP CheckWorkstepDone:   // S19, max time T#10S, warning time T#7S
              N    #txCheckWorkStep
   END_STEP
   TRANSITION WorkstepDone FROM CheckWorkstepDone TO IndexerHomePos   // T21
      := NOT #releaseWorkStep AND #qxCarrierIsDone;
   END_TRANSITION
   TRANSITION NotDone FROM CheckWorkstepDone TO JogS1   // T22, jump
      := #CheckWorkstepDone.T >= t#1s;
   END_TRANSITION
   STEP Release:   // S20, max time T#10S, warning time T#7S
          S1  S    #releaseWorkStep
   END_STEP
   TRANSITION WorkstepIsReleased FROM Release TO JogS1   // T23
      := true;
   END_TRANSITION
   STEP Warte_Endziel_frei:   // S21, max time T#10S, warning time T#7S
   END_STEP
   TRANSITION EndzielFrei FROM Warte_Endziel_frei TO OpenStopper   // T24
      := (NOT #ixTargetReached OR NOT #ixCheckTargetReached) AND #ixReleaseTransfer;
   END_TRANSITION
   TRANSITION EndzielNichtFrei FROM Warte_Endziel_frei TO JogS2   // T25, jump
      := #Warte_Endziel_frei.T >= t#3s;
   END_TRANSITION

   // permanent post-instructions
   NETWORK 1
   TITLE = Störungssignal weitergeben
      #sq.error := #ERR_FLT;
   NETWORK 2
   TITLE = Ablauf ist aktiv
      #qxIsActive := #sq.running;
   NETWORK 3
   TITLE = steht in Grundstellung
      #qxIsInHome := #sq.inHome AND NOT #sq.running;
   NETWORK 4
   TITLE = WT-Träger ist fertig bearbeitet worden
      IF NOT #releaseWorkStep AND #txCheckWorkStep THEN #qxCarrierIsDone := TRUE; END_IF;
END_FUNCTION_BLOCK

// folder: 9. Library/9.4 HMI

FUNCTION_BLOCK "HmiManualMovementController"   // FB9401, SCL
{ S7_Optimized_Access := 'TRUE' }
VERSION : 0.1
   VAR_INPUT
      showRows : USInt := 4;
   END_VAR
   VAR_IN_OUT
      manualMovements : "typeManualMovements";
      hmiManualMovement : "typeHmiManualMovement";
   END_VAR
   VAR
      susiFirstRowManualMoveNo : USInt;
      susiLastRowManualMoveNo : USInt;
      susiSelectedStationOld : USInt;
      susiSelectedStationHasChanged : Bool;
      sinstTonShowSymbols : TON_TIME;
   END_VAR
   VAR_TEMP
      tusiRows : USInt;   // Index variable hmi rows
      tusiMM : USInt;   // Index variable manual move
      tusiOffset : USInt;
      txResetShowSymbols : Bool;
      tuiOffsetShowSymbols : UInt;
   END_VAR
BEGIN
   // Ersteller: Andreas Fast Automation
   // E-Mail: automation@fast-andreas.de
   //
   // Projekt dient zu Demonstrationszwecken und frei genutzt werden.
   //
   // Bausteinbeschreibung:
   // 

   // Check selected station has changed
   #susiSelectedStationHasChanged := false;
   IF #hmiManualMovement.selection.station <> #susiSelectedStationOld THEN
       #susiFirstRowManualMoveNo := 0;
       #susiLastRowManualMoveNo := 0;
       #hmiManualMovement.selection.page := 0;
       #hmiManualMovement.selection.ofMaxPages := 0;
       #susiSelectedStationHasChanged := true;

       // Initialise rows on changed selected station
       FOR #tusiRows := 1 TO "SYS_HMI_SETUPMAXROWS" DO
           #hmiManualMovement.rows[#tusiRows].move := #manualMovements.movements[0];
           #hmiManualMovement.rows[#tusiRows].movementNo := 0;
           #hmiManualMovement.rows[#tusiRows].textlistFunctionName := 0;
           #hmiManualMovement.rows[#tusiRows].textlistFunctionExecuteLeft := 0;
           #hmiManualMovement.rows[#tusiRows].textlistFunctionFinalPosLeft := 0;
           #hmiManualMovement.rows[#tusiRows].textlistFunctionExecuteRight := 0;
           #hmiManualMovement.rows[#tusiRows].textlistFunctionFinalPosRight := 0;

       END_FOR;




   END_IF;
   #susiSelectedStationOld := #hmiManualMovement.selection.station;

   // Manage manual movement rows on HMI
   IF #hmiManualMovement.selection.station > 0 THEN

       // Find first and last manual movement number of selected station
       IF #susiSelectedStationHasChanged THEN
           #susiSelectedStationHasChanged := false;

           FOR #tusiMM := 1 TO "SYS_MANUALMOVEMENTS" DO
               // Check if the selected station is the same in manual movements (find the first manual movement of selected station)
               IF #manualMovements.movements[#tusiMM].attributes.stationNo = #hmiManualMovement.selection.station THEN
                   #susiFirstRowManualMoveNo := #tusiMM;
                   #susiLastRowManualMoveNo := #tusiMM;
                   #hmiManualMovement.selection.page := 1;
                   EXIT;
               END_IF;
           END_FOR;

           FOR #tusiMM := #susiLastRowManualMoveNo + 1 TO "SYS_MANUALMOVEMENTS" DO
               // Check if the selected station is not the same anymore in manual movements
               IF #manualMovements.movements[#tusiMM].attributes.stationNo <> #hmiManualMovement.selection.station THEN
                   EXIT;
               END_IF;
               // Check if the movement is visible (not reserved), otherwise don't change LastRow-Variable
               IF #manualMovements.movements[#tusiMM].attributes.showName THEN
                   #susiLastRowManualMoveNo := #tusiMM;
               END_IF;
           END_FOR;

       END_IF;

       IF #susiFirstRowManualMoveNo > 0 THEN // Control displayed page

           #hmiManualMovement.selection.ofMaxPages := (#susiLastRowManualMoveNo - #susiFirstRowManualMoveNo + 1) / #showRows;
           IF FRAC(INT_TO_REAL((#susiLastRowManualMoveNo - #susiFirstRowManualMoveNo + 1)) / #showRows) > 0.0 THEN
               #hmiManualMovement.selection.ofMaxPages += 1;
           END_IF;
           // Next page
           IF #hmiManualMovement.selection.nextPage THEN
               #hmiManualMovement.selection.nextPage := false;
               IF #hmiManualMovement.selection.page >= #hmiManualMovement.selection.ofMaxPages THEN
                   #hmiManualMovement.selection.page := 1;
               ELSE
                   #hmiManualMovement.selection.page += 1;
               END_IF;
           END_IF;
           // Previous page
           IF #hmiManualMovement.selection.previousPage THEN
               #hmiManualMovement.selection.previousPage := false;
               IF #hmiManualMovement.selection.page <= 1 THEN
                   #hmiManualMovement.selection.page := #hmiManualMovement.selection.ofMaxPages;
               ELSE
                   #hmiManualMovement.selection.page -= 1;
               END_IF;
           END_IF;
       END_IF;


       IF #susiFirstRowManualMoveNo > 0 THEN
           // Connect manual movements to hmi rows
           FOR #tusiRows := 1 TO "SYS_HMI_SETUPMAXROWS" DO
               #tusiOffset := #tusiRows - 1 + (#hmiManualMovement.selection.page-1) * #showRows;

               // Check max configured rows for HMI is reached
               IF #showRows < #tusiRows THEN
                   EXIT;
               END_IF;

               // Connect manual movements to HMI rows
               IF #susiFirstRowManualMoveNo + #tusiOffset <= #susiLastRowManualMoveNo THEN 
                   // Manual Movements -> HMI
                   #hmiManualMovement.rows[#tusiRows].movementNo := #susiFirstRowManualMoveNo + #tusiOffset;
                   #hmiManualMovement.rows[#tusiRows].move.attributes := #manualMovements.movements[#susiFirstRowManualMoveNo + #tusiOffset].attributes;
                   #hmiManualMovement.rows[#tusiRows].move.control.value := #manualMovements.movements[#susiFirstRowManualMoveNo + #tusiOffset].control.value;
                   #hmiManualMovement.rows[#tusiRows].move.control.homeAct := #manualMovements.movements[#susiFirstRowManualMoveNo + #tusiOffset].control.homeAct;
                   #hmiManualMovement.rows[#tusiRows].move.control.workAct := #manualMovements.movements[#susiFirstRowManualMoveNo + #tusiOffset].control.workAct;
                   #hmiManualMovement.rows[#tusiRows].move.control.homeIsInterlocked := #manualMovements.movements[#susiFirstRowManualMoveNo + #tusiOffset].control.homeIsInterlocked;
                   #hmiManualMovement.rows[#tusiRows].move.control.workIsInterlocked := #manualMovements.movements[#susiFirstRowManualMoveNo + #tusiOffset].control.workIsInterlocked;
                   #hmiManualMovement.rows[#tusiRows].move.control.inHomePos := #manualMovements.movements[#susiFirstRowManualMoveNo + #tusiOffset].control.inHomePos;
                   #hmiManualMovement.rows[#tusiRows].move.control.inWorkPos := #manualMovements.movements[#susiFirstRowManualMoveNo + #tusiOffset].control.inWorkPos;

                   // HMI -> Manual Movements 
                   #manualMovements.movements[#susiFirstRowManualMoveNo + #tusiOffset].control.moveHomePos := #hmiManualMovement.rows[#tusiRows].move.control.moveHomePos;
                   #manualMovements.movements[#susiFirstRowManualMoveNo + #tusiOffset].control.moveWorkPos := #hmiManualMovement.rows[#tusiRows].move.control.moveWorkPos;

                   // Update textlist values
                   IF #hmiManualMovement.selection.showSymbols THEN
                       #tuiOffsetShowSymbols := 1;
                   ELSE
                       #tuiOffsetShowSymbols := 0;
                   END_IF;
                   #hmiManualMovement.rows[#tusiRows].textlistFunctionName := USINT_TO_UINT(#hmiManualMovement.rows[#tusiRows].movementNo) * 10 + #tuiOffsetShowSymbols;
                   #hmiManualMovement.rows[#tusiRows].textlistFunctionExecuteLeft := USINT_TO_UINT(#hmiManualMovement.rows[#tusiRows].movementNo) * 10 + 2 + #tuiOffsetShowSymbols;
                   #hmiManualMovement.rows[#tusiRows].textlistFunctionFinalPosLeft := USINT_TO_UINT(#hmiManualMovement.rows[#tusiRows].movementNo) * 10 + 4 + #tuiOffsetShowSymbols;
                   #hmiManualMovement.rows[#tusiRows].textlistFunctionExecuteRight := USINT_TO_UINT(#hmiManualMovement.rows[#tusiRows].movementNo) * 10 + 6 + #tuiOffsetShowSymbols;
                   #hmiManualMovement.rows[#tusiRows].textlistFunctionFinalPosRight := USINT_TO_UINT(#hmiManualMovement.rows[#tusiRows].movementNo) * 10 + 8 + #tuiOffsetShowSymbols;

               ELSE
                   #hmiManualMovement.rows[#tusiRows].move := #manualMovements.movements[0];
                   #hmiManualMovement.rows[#tusiRows].movementNo := 0;
                   #hmiManualMovement.rows[#tusiRows].textlistFunctionName := 0;
                   #hmiManualMovement.rows[#tusiRows].textlistFunctionExecuteLeft := 0;
                   #hmiManualMovement.rows[#tusiRows].textlistFunctionFinalPosLeft := 0;
                   #hmiManualMovement.rows[#tusiRows].textlistFunctionExecuteRight := 0;
                   #hmiManualMovement.rows[#tusiRows].textlistFunctionFinalPosRight := 0;
               END_IF;


           END_FOR;
       END_IF; 

   ELSE
       #hmiManualMovement.selection.nextPage := false;
       #hmiManualMovement.selection.previousPage := false;
   END_IF;


   // Deactivate show symbols
   #sinstTonShowSymbols(IN := #hmiManualMovement.selection.showSymbols,
                        PT := t#30s,
                        Q => #txResetShowSymbols);

   IF #txResetShowSymbols OR #susiSelectedStationHasChanged THEN
       #hmiManualMovement.selection.showSymbols := false;
   END_IF;
END_FUNCTION_BLOCK

FUNCTION_BLOCK "HmiShowStepSequences"   // FB9402, SCL
{ S7_Optimized_Access := 'TRUE' }
VERSION : 0.1
   VAR_INPUT
      iusiStation : USInt;
      iusiSequence : USInt;
   END_VAR
   VAR_OUTPUT
      qudtStepSeqs : "typeStepSequence";
   END_VAR
   VAR
      susiStationOld : USInt;
   END_VAR
BEGIN
   // Ersteller: Andreas Fast Automation
   // E-Mail: automation@fast-andreas.de
   //
   // Projekt dient zu Demonstrationszwecken und frei genutzt werden.
   //
   // Bausteinbeschreibung:
   // 

   IF #iusiStation <> #susiStationOld THEN

       #qudtStepSeqs := "Machine".stations.station[#iusiStation].stepSeqs.stepSeq[#iusiSequence];

   END_IF;
   #susiStationOld := #iusiStation;
END_FUNCTION_BLOCK

// folder: 9. Library/9.9 Templates

FUNCTION_BLOCK "StepSequence"   // FB992, GRAPH_PLUS
{ S7_Optimized_Access := 'TRUE' }
VERSION : 0.1
   VAR_INPUT
      OFF_SQ : Bool := false;   // Kette ausschalten
      INIT_SQ : Bool := false;   // Kette in Initialzustand versetzen
      ACK_EF : Bool := false;   // Alle Fehler und Störungen quittieren
      S_PREV : Bool := false;   // Vorherigen Schritt am Parameter S_NO ausgeben
      S_NEXT : Bool := false;   // Nächsten Schritt am Parameter S_NO anzeigen
      SW_AUTO : Bool := false;   // Automatischer Betrieb
      SW_TAP : Bool := false;   // Halbautomatisch/Weiterschalten mit Transition
      SW_TOP : Bool := false;   // Halbautomatisch/Ignoriere Transition
      SW_MAN : Bool := false;   // Handbetrieb
      S_SEL : Int := 0;   // Schritt auswählen, der an S_NO ausgegeben werden soll
      S_ON : Bool := false;   // Schritt aktivieren, der an Parameter S_NO anliegt
      S_OFF : Bool := false;   // Schritt deaktivieren, der an Parameter S_NO anliegt
      T_PUSH : Bool := false;   // Schaltfreigabe für Transition im halbautomatischen Betrieb
   END_VAR
   VAR_OUTPUT
      S_NO : Int := 0;   // Schrittnummer
      S_MORE : Bool := false;   // Weitere Schritte sind vorhanden und können in S_NO angezeigt werden.
      S_ACTIVE : Bool := false;   // Schritt, der an Parameter S_NO angezeigt wird, ist aktiv
      ERR_FLT : Bool := false;   // Sammelfehler Interlock oder Supervision
      AUTO_ON : Bool := false;   // Automatischer Betrieb eingeschaltet
      TAP_ON : Bool := false;   // Halbautomatischer Betrieb/Schritt mit Transition eingeschaltet
      TOP_ON : Bool := false;   // Halbautomatischer Betrieb/Ignoriere Transition eingeschaltet
      MAN_ON : Bool := false;   // Handbetrieb eingeschaltet
   END_VAR
   VAR_IN_OUT
      signals : "typeStationSignals";   // Stationssteuersignale
      sq : "typeStepSequence";   // Schrittkettensteuersignale
   END_VAR
   VAR
      startCondition : Bool;   // Startbedingung
      HMI_INFO : Array[0..8] of UInt;
      IF_PAR : G7_IfParPlus_V6;
      RT_DATA : G7_RTDataPlus_V6;   // Interner Datenbereich
      Automatikablauf : G7_TransitionPlus_V6;   // Transitionsstruktur
      Freigabe : G7_TransitionPlus_V6;   // Transitionsstruktur
      Trans3 : G7_TransitionPlus_V6;   // Transitionsstruktur
      Fertig : G7_TransitionPlus_V6;   // Transitionsstruktur
      Grundstellungsfahrt : G7_TransitionPlus_V6;   // Transitionsstruktur
      GST_Aktiv : G7_TransitionPlus_V6;   // Transitionsstruktur
      GST_Beendet : G7_TransitionPlus_V6;   // Transitionsstruktur
      Beendet : G7_TransitionPlus_V6;   // Transitionsstruktur
      Initialschritt : G7_StepPlus_V6;   // Schrittstruktur
      Grundstellung : G7_StepPlus_V6;   // Schrittstruktur
      Ablauf : G7_StepPlus_V6;   // Schrittstruktur
      Fertigmeldung : G7_StepPlus_V6;   // Schrittstruktur
      "Start Grundstellungsfahrt" : G7_StepPlus_V6;   // Schrittstruktur
      "Fertig Grundstellungsfahrt" : G7_StepPlus_V6;   // Schrittstruktur
      Ende : G7_StepPlus_V6;   // Schrittstruktur
      SINI : Array[0..1] of USInt;
      LSTT : Array[0..7] of USInt;
      ATAJ : Array[0..7] of USInt;
      ATAB : Array[0..7] of USInt;
      PSTT : Array[0..7] of USInt;
      NSTT : Array[0..7] of USInt;
      ASSJ : Array[0..6] of USInt;
      ASSB : Array[0..6] of USInt;
      PTTS : Array[0..6] of USInt;
      NTTS : Array[0..6] of USInt;
      SW_SQTS : Array[0..6] of USInt;
      SWITCH : Array[0..1] of USInt;
      TVX : Array[0..3] of USInt;
      TTX : Array[0..3] of USInt;
      TSX : Array[0..1] of USInt;
      S00X : Array[0..1] of USInt;
      SOFFX : Array[0..1] of USInt;
      SONX : Array[0..1] of USInt;
      SAX : Array[0..1] of USInt;
      SERRX : Array[0..7] of USInt;
      SMX : Array[0..7] of USInt;
      S0X : Array[0..7] of USInt;
      S1X : Array[0..7] of USInt;
      IL_ALARM_INST : Diag_Alarm;
      SUP_ALARM_INST : Diag_Alarm;
      STEP_TIME_ALARM_INST : Diag_Alarm;
      IEC_TIMER_INST : IEC_TIMER;
      TRANSACTION_FLAG : Bool := false;
   END_VAR
   // SINI[0] := 2;
   // LSTT[0] := 255;
   // LSTT[1] := 255;
   // LSTT[2] := 255;
   // LSTT[3] := 255;
   // LSTT[4] := 255;
   // LSTT[5] := 255;
   // LSTT[6] := 255;
   // LSTT[7] := 1;
   // ATAJ[1] := 1;
   // ATAJ[2] := 2;
   // ATAJ[3] := 6;
   // ATAJ[4] := 4;
   // ATAJ[5] := 5;
   // ATAJ[6] := 3;
   // ATAJ[7] := 7;
   // ATAB[0] := 4;
   // ATAB[1] := 1;
   // ATAB[2] := 2;
   // ATAB[3] := 3;
   // ATAB[5] := 5;
   // ATAB[6] := 6;
   // ATAB[7] := 7;
   // PSTT[1] := 1;
   // PSTT[2] := 2;
   // PSTT[3] := 3;
   // PSTT[5] := 4;
   // PSTT[6] := 5;
   // PSTT[7] := 6;
   // NSTT[0] := 1;
   // NSTT[1] := 2;
   // NSTT[2] := 3;
   // NSTT[3] := 6;
   // NSTT[4] := 4;
   // NSTT[5] := 5;
   // NSTT[6] := 6;
   // NSTT[7] := 1;
   // ASSJ[1] := 1;
   // ASSJ[2] := 2;
   // ASSJ[3] := 3;
   // ASSJ[4] := 4;
   // ASSJ[5] := 5;
   // ASSJ[6] := 6;
   // ASSB[1] := 1;
   // ASSB[2] := 2;
   // ASSB[3] := 3;
   // ASSB[4] := 4;
   // ASSB[5] := 5;
   // ASSB[6] := 6;
   // PTTS[0] := 255;
   // PTTS[2] := 1;
   // PTTS[3] := 2;
   // PTTS[4] := 4;
   // PTTS[5] := 5;
   // PTTS[6] := 3;
   // NTTS[1] := 1;
   // NTTS[2] := 2;
   // NTTS[3] := 3;
   // NTTS[4] := 5;
   // NTTS[5] := 6;
   // NTTS[6] := 7;
   // SW_SQTS[1] := 1;
   // SW_SQTS[2] := 1;
   // SW_SQTS[3] := 1;
   // SW_SQTS[4] := 2;
   // SW_SQTS[5] := 2;
   // SW_SQTS[6] := 3;
   // TVX[0] := 16#1;
   // TTX[0] := 16#1;
   // TSX[0] := 16#1;
   // S00X[0] := 16#1;
   // SOFFX[0] := 16#1;
   // SONX[0] := 16#1;
   // SAX[0] := 16#1;
   // SERRX[0] := 16#1;
   // SMX[0] := 16#1;
   // S0X[0] := 16#1;
   // S1X[0] := 16#1;
BEGIN
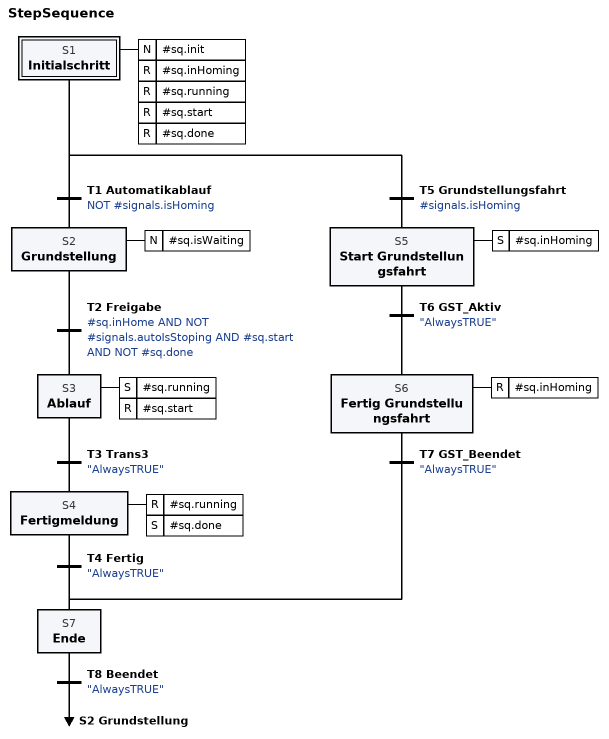
   // permanent pre-instructions
   NETWORK 1
   TITLE = Schrittkette in Grundstellung
      #sq.inHome := #Grundstellung.X;
   NETWORK 2
   TITLE = Schrittkette starten
      IF #sq.inHome AND NOT #sq.running AND #signals.releaseCycle AND NOT #signals.isHoming AND #startCondition THEN
          #sq.start := TRUE;
          #sq.done := FALSE;
      END_IF;

   // sequencer 1
   INITIAL_STEP Initialschritt:   // S1, max time T#10S, warning time T#7S
              N    #sq.init
              R    #sq.inHoming
              R    #sq.running
              R    #sq.start
              R    #sq.done
   END_STEP
   TRANSITION Automatikablauf FROM Initialschritt TO Grundstellung   // T1
      := NOT #signals.isHoming;
   END_TRANSITION
   TRANSITION Grundstellungsfahrt FROM Initialschritt TO "Start Grundstellungsfahrt"   // T5
      := #signals.isHoming;
   END_TRANSITION
   STEP Grundstellung:   // S2, max time T#10S, warning time T#7S
              N    #sq.isWaiting
   END_STEP
   TRANSITION Freigabe FROM Grundstellung TO Ablauf   // T2
      := #sq.inHome AND NOT #signals.autoIsStoping AND #sq.start AND NOT #sq.done;
   END_TRANSITION
   STEP Ablauf:   // S3, max time T#10S, warning time T#7S
              S    #sq.running
              R    #sq.start
   END_STEP
   TRANSITION Trans3 FROM Ablauf TO Fertigmeldung   // T3
      := "AlwaysTRUE";
   END_TRANSITION
   STEP Fertigmeldung:   // S4, max time T#10S, warning time T#7S
              R    #sq.running
              S    #sq.done
   END_STEP
   TRANSITION Fertig FROM Fertigmeldung TO Ende   // T4
      := "AlwaysTRUE";
   END_TRANSITION
   STEP "Start Grundstellungsfahrt":   // S5, max time T#10S, warning time T#7S
              S    #sq.inHoming
   END_STEP
   TRANSITION GST_Aktiv FROM "Start Grundstellungsfahrt" TO "Fertig Grundstellungsfahrt"   // T6
      := "AlwaysTRUE";
   END_TRANSITION
   STEP "Fertig Grundstellungsfahrt":   // S6, max time T#10S, warning time T#7S
              R    #sq.inHoming
   END_STEP
   TRANSITION GST_Beendet FROM "Fertig Grundstellungsfahrt" TO Ende   // T7
      := "AlwaysTRUE";
   END_TRANSITION
   STEP Ende:   // S7, max time T#10S, warning time T#7S
   END_STEP
   TRANSITION Beendet FROM Ende TO Grundstellung   // T8, jump
      := "AlwaysTRUE";
   END_TRANSITION

   // permanent post-instructions
   NETWORK 1
   TITLE = Störungssignal weitergeben
      #sq.error := #ERR_FLT;
END_FUNCTION_BLOCK

(* ===== HMI "HMI_RT_1" =====
system functions are stored by id; their names below are inferred from use
connection "HMI_Verbindung_1": ETHERNET, S7_1500_OMS

HMI tags "Standard-Variablentabelle"
   "Header_Line_1" : UInt, internal
   "Header_Line_2" : UInt, internal

HMI tags "Einrichtfunktionen"
   "HmiManualMovement_selection_station" : USInt = PLC HmiManualMovement.selection.station AT %DB1.DBX0.0, 1 s
   "HmiManualMovement_selection_page" : USInt = PLC HmiManualMovement.selection.page AT %DB1.DBB0, 1 s
   "HmiManualMovement_selection_ofMaxPages" : USInt = PLC HmiManualMovement.selection.ofMaxPages AT %DB1.DBB0, 1 s
   "HmiManualMovement_selection_nextPage" : Bool = PLC HmiManualMovement.selection.nextPage AT %DB1.DBB0, 1 s
   "HmiManualMovement_selection_previousPage" : Bool = PLC HmiManualMovement.selection.previousPage AT %DB1.DBX0.0, 1 s
   "HmiManualMovement_selection_showSymbols" : Bool = PLC HmiManualMovement.selection.showSymbols AT %DB1.DBX0.0, 1 s
   "HmiManualMovement_rows{1}" : typeHmiManualMove = PLC HmiManualMovement.rows[1] AT %DB1.DBX0.0, 100 ms
   "HmiManualMovement_rows{2}" : typeHmiManualMove = PLC HmiManualMovement.rows[2] AT %DB1.DBW0, 100 ms
   "HmiManualMovement_rows{3}" : typeHmiManualMove = PLC HmiManualMovement.rows[3] AT %DB1.DBW0, 100 ms
   "HmiManualMovement_rows{4}" : typeHmiManualMove = PLC HmiManualMovement.rows[4] AT %DB1.DBW0, 100 ms

HMI tags "Alarmserver"
   "Alarmserver_hmi_machine" : typeHmiErrMsg = PLC Alarmserver.hmi.machine AT %DB1.DBW0, 1 s

HMI tags "Stationen"
   "Machine_stations_station{1}" : typeStation = PLC Machine.stations.station[1] AT %DB1.DBW0, 1 s
   "Machine_stations_station{2}" : typeStation = PLC Machine.stations.station[2] AT %DB1.DBW0, 1 s
   "Machine_stations_station{3}" : typeStation = PLC Machine.stations.station[3] AT %DB1.DBW0, 1 s
   "Machine_stations_station{4}" : typeStation = PLC Machine.stations.station[4] AT %DB1.DBW0, 1 s
   "Machine_stations_station{5}" : typeStation = PLC Machine.stations.station[5] AT %DB1.DBW0, 1 s
   "Machine_stations_station{10}" : typeStation = PLC Machine.stations.station[10] AT %DB1.DBW0, 1 s
   "Machine_machine" : typeMachine = PLC Machine.machine AT %DB1.DBW0, 1 s
   "Machine_stations_station{6}" : typeStation = PLC Machine.stations.station[6] AT %DB1.DBW0, 1 s
   "Machine_stations_station{7}" : typeStation = PLC Machine.stations.station[7] AT %DB1.DBW0, 1 s
   "Machine_stations_station{8}" : typeStation = PLC Machine.stations.station[8] AT %DB1.DBW0, 1 s
   "Machine_stations_station{9}" : typeStation = PLC Machine.stations.station[9] AT %DB1.DBW0, 1 s

HMI tags "Interne Variablen"
   "Übersicht_Station1" : Int, internal
   "Übersicht_Station2" : Int, internal
   "Übersicht_Station3" : Int, internal
   "Übersicht_Station4" : Int, internal
   "Übersicht_Station5" : Int, internal
   "Übersicht_Station6" : Int, internal
   "Übersicht_Station7" : Int, internal
   "Übersicht_Station8" : Int, internal
   "Übersicht_Station9" : Int, internal
   "Übersicht_Station10" : Int, internal

discrete alarms
   1001: 'Maschine Störung 1: Initialisierung für die Einrichtbewegungen ist fehlerhaft', class Errors, trigger "alarmAckPlc" bit 0
   1002: 'Maschine Störung 2: Not-Aus aktiv', class Errors, trigger "alarmAckPlc" bit 1
   1003: 'Maschine Störung 3', class Errors, trigger "alarmAckPlc" bit 2
   1004: 'Maschine Störung 4', class Errors, trigger "alarmAckPlc" bit 3
   1005: 'Maschine Störung', class Errors, trigger "alarmAckPlc" bit 4
   1006: 'Maschine Störung 6', class Errors, trigger "alarmAckPlc" bit 5
   1007: 'Maschine Störung 7', class Errors, trigger "alarmAckPlc" bit 6
   1008: 'Maschine Störung 8', class Errors, trigger "alarmAckPlc" bit 7
   1009: 'Maschine Störung 9', class Errors, trigger "alarmAckPlc" bit 8
   1010: 'Maschine Störung 10', class Errors, trigger "alarmAckPlc" bit 9
   1011: 'Maschine Störung 11', class Errors, trigger "alarmAckPlc" bit 10
   1012: 'Maschine Störung 12', class Errors, trigger "alarmAckPlc" bit 11
   1013: 'Maschine Störung 13', class Errors, trigger "alarmAckPlc" bit 12
   1014: 'Maschine Störung 14', class Errors, trigger "alarmAckPlc" bit 13
   1015: 'Maschine Störung 15', class Errors, trigger "alarmAckPlc" bit 14
   1016: 'Maschine Störung 16', class Errors, trigger "alarmAckPlc" bit 15
   1017: 'Maschine Störung 17', class Errors, trigger "alarmAckPlc" bit 16
   1018: 'Maschine Störung 18', class Errors, trigger "alarmAckPlc" bit 17
   1019: 'Maschine Störung 19', class Errors, trigger "alarmAckPlc" bit 18
   1020: 'Maschine Störung 20', class Errors, trigger "alarmAckPlc" bit 19
   1021: 'Maschine Störung 21', class Errors, trigger "alarmAckPlc" bit 20
   1022: 'Maschine Störung 22', class Errors, trigger "alarmAckPlc" bit 21
   1023: 'Maschine Störung 23', class Errors, trigger "alarmAckPlc" bit 22
   1024: 'Maschine Störung 24', class Errors, trigger "alarmAckPlc" bit 23
   1025: 'Maschine Störung 25', class Errors, trigger "alarmAckPlc" bit 24
   1026: 'Maschine Störung 26', class Errors, trigger "alarmAckPlc" bit 25
   1027: 'Maschine Störung 27', class Errors, trigger "alarmAckPlc" bit 26
   1028: 'Maschine Störung 28', class Errors, trigger "alarmAckPlc" bit 27
   1029: 'Maschine Störung 29', class Errors, trigger "alarmAckPlc" bit 28
   1030: 'Maschine Störung 30', class Errors, trigger "alarmAckPlc" bit 29
   1031: 'Maschine Störung 31', class Errors, trigger "alarmAckPlc" bit 30
   1032: 'Maschine Störung 32', class Errors, trigger "alarmAckPlc" bit 31
   1: 'Maschine ist ausgeschaltet', class Warnings, trigger "message" bit 0
   2: 'Maschine: Handbetrieb aktiv', class Warnings, trigger "message" bit 1
   3: 'Maschine: Meldungstext', class Warnings, trigger "message" bit 2
   4: 'Maschine: Meldungstext', class Warnings, trigger "message" bit 3
   31: 'Maschine: Meldungstext', class Warnings, trigger "message" bit 31
   30: 'Maschine: Meldungstext', class Warnings, trigger "message" bit 30
   5: 'Maschine: Meldungstext', class Warnings, trigger "message" bit 5
   6: 'Maschine: Meldungstext', class Warnings, trigger "message" bit 6
   7: 'Maschine: Meldungstext', class Warnings, trigger "message" bit 7
   8: 'Maschine: Meldungstext', class Warnings, trigger "message" bit 8
   9: 'Maschine: Meldungstext', class Warnings, trigger "message" bit 9
   10: 'Maschine: Meldungstext', class Warnings, trigger "message" bit 10
   11: 'Maschine: Meldungstext', class Warnings, trigger "message" bit 11
   12: 'Maschine: Meldungstext', class Warnings, trigger "message" bit 12
   13: 'Maschine: Meldungstext', class Warnings, trigger "message" bit 13
   14: 'Maschine: Meldungstext', class Warnings, trigger "message" bit 14
   15: 'Maschine: Meldungstext', class Warnings, trigger "message" bit 15
   16: 'Maschine: Meldungstext', class Warnings, trigger "message" bit 16
   17: 'Maschine: Meldungstext', class Warnings, trigger "message" bit 17
   18: 'Maschine: Meldungstext', class Warnings, trigger "message" bit 18
   19: 'Maschine: Meldungstext', class Warnings, trigger "message" bit 19
   20: 'Maschine: Meldungstext', class Warnings, trigger "message" bit 20
   21: 'Maschine: Meldungstext', class Warnings, trigger "message" bit 21
   22: 'Maschine: Meldungstext', class Warnings, trigger "message" bit 22
   23: 'Maschine: Meldungstext', class Warnings, trigger "message" bit 23
   24: 'Maschine: Meldungstext', class Warnings, trigger "message" bit 24
   25: 'Maschine: Meldungstext', class Warnings, trigger "message" bit 25
   26: 'Maschine: Meldungstext', class Warnings, trigger "message" bit 26
   27: 'Maschine: Meldungstext', class Warnings, trigger "message" bit 27
   28: 'Maschine: Meldungstext', class Warnings, trigger "message" bit 28
   29: 'Maschine: Meldungstext', class Warnings, trigger "message" bit 29

text list "Header_Line_1": 1 'Grundbild'; 100 'Automatik'; 10 'Einrichten'; 12 'Einrichtfunktionen'; 1000 'Systembilder / System screens'; 1001 'SIMATIC PLC Systemdiagnose / SIMATIC PLC system diagnostics'; 1002 'Projektinformationen / Project information'; 1003 'Systemeinstellungen / System settings'; 1004 'Benutzerverwaltung / User administration'; 1005 'Systeminformationen / System information'; 1006 'Verschiedene Aufgaben / Different jobs'; 2 'Übersicht'

